Yaskawa INFORM job: SKRZYNIA_5140_180_STOPNI_10B_NEW.JBI

/JOB
//NAME SKRZYNIA_5140_180_STOPNI_10B_NEW
///FOLDERNAME 02-SKRZYNIE_JOBS
//POS
///NPOS 714,714,0,30,0,0
///TOOL 0
///POSTYPE PULSE
///PULSE
C00000=-21231,-51303,42314,2367,6591,-1439
C00001=-12854,-61498,-6635,149088,-29435,16513
C00002=84284,-61498,-6635,149088,14842,16513
C00003=84426,-61498,-62039,149088,14842,16513
C00004=84426,-61498,-83719,149088,14842,16513
C00005=40079,-25830,-61904,72398,37828,17494
C00006=40079,-25830,-61904,72398,37828,17494
C00007=38824,-23395,-60038,72349,38727,17731
C00008=41545,-22667,-59464,70826,37145,18191
C00009=40079,-25830,-61904,72398,37828,17494
C00010=40079,-23879,-31232,97616,36989,2612
C00011=40241,-22903,-30855,97033,36795,2952
C00012=39596,-21803,-29985,96678,37187,3182
C00013=41542,-21522,-29763,96797,35874,3054
C00014=40241,-22903,-30855,97033,36795,2952
C00015=44500,-22967,-34027,49689,40772,15208
C00016=44759,-21950,-33222,49364,40770,15399
C00017=43898,-20603,-32137,49608,41392,15289
C00018=45676,-20288,-31878,48567,40497,15854
C00019=44759,-21950,-33222,49364,40770,15399
C00020=50639,-31838,-53853,40430,42590,20636
C00021=47737,-42531,-47731,84740,46626,-3202
C00022=73324,-51450,-15857,136644,48513,-27329
C00023=28578,-31257,-33285,101874,54895,-3139
C00024=29101,-23166,-41439,93785,52323,3372
C00025=30342,-16402,-40775,90158,51109,6027
C00026=29555,-14242,-38855,90054,51607,6222
C00027=31304,-14182,-38798,89754,50458,6198
C00028=30342,-16402,-40775,90158,51109,6027
C00029=37840,-26567,-47806,97824,39338,5403
C00030=38314,-22656,-45541,96192,38787,6352
C00031=38740,-21749,-44817,95954,38481,6451
C00032=38106,-20505,-43805,95701,38856,6673
C00033=39920,-20274,-43616,95549,37666,6573
C00034=38740,-21749,-44817,95954,38481,6451
C00035=35154,-23288,-28184,89821,43405,2441
C00036=35403,-21021,-26397,89340,43215,2751
C00037=34678,-19569,-25213,89063,43699,2948
C00038=36545,-19419,-25091,89018,42427,2940
C00039=35403,-21021,-26397,89340,43215,2751
C00040=46673,-28267,-59493,36306,49500,22578
C00041=47298,-25083,-54483,36432,48421,22382
C00042=46134,-23276,-53085,36983,49197,22170
C00043=48093,-22778,-52692,35651,48513,22818
C00044=47298,-25083,-54483,36432,48421,22382
C00045=43000,-32780,-49011,53703,41088,15214
C00046=66148,-65994,-55487,105361,28212,-7739
C00047=66148,-65994,-55487,105361,28212,-7739
C00048=59848,-54778,-49507,133915,29212,-10807
C00049=45497,-38347,-41839,114412,32622,-465
C00050=46376,-32635,-46933,102993,29107,5780
C00051=46303,-28031,-46898,97061,28371,8976
C00052=45038,-26161,-45521,96183,29128,9541
C00053=46946,-25787,-45238,96120,27855,9431
C00054=46303,-28031,-46898,97061,28371,8976
C00055=45864,-17128,1685,129467,40696,-9274
C00056=46023,-15894,1830,128891,40053,-8896
C00057=45181,-14790,2774,128176,40341,-8535
C00058=46921,-14545,2986,129317,39465,-9073
C00059=45402,-17127,796,128656,40504,-8810
C00060=42828,-21985,-11573,106778,34538,-1929
C00061=43349,-21404,-11124,106831,34165,-1930
C00062=42250,-19876,-9917,105946,34757,-1485
C00063=44494,-19460,-9583,106781,33302,-1837
C00064=42797,-21858,-11474,106726,34550,-1903
C00065=42956,-14057,7354,88292,32197,-569
C00066=43438,-13569,7781,88275,31880,-510
C00067=42549,-12302,8904,87823,32462,-349
C00068=44721,-11883,9282,88161,31033,-316
C00069=42944,-14884,6642,88491,32210,-682
C00070=72417,-64226,-72669,53660,37323,27470
C00071=81480,-74508,-67932,111005,17511,3722
C00072=42492,-36415,-29790,92406,42740,11684
C00073=29699,-14901,-14062,86637,51249,15251
C00074=28921,-12904,-12269,86425,51786,15406
C00075=30978,-12767,-12144,86426,50380,15429
C00076=29506,-17416,-16239,86937,51377,15018
C00077=88410,-69609,-60867,139529,19008,-8209
C00078=82254,-59190,-37505,135829,26015,-2584
C00079=48709,-26647,-10027,118963,31871,904
C00080=44740,-24992,-19428,105622,30913,8023
C00081=35836,-10089,175,120717,54219,3716
C00082=33571,-11609,-5533,116057,52820,8482
C00083=32638,-9483,-3533,115639,53262,8773
C00084=34483,-9329,-3384,116184,52162,8425
C00085=33571,-11609,-5533,116057,52820,8482
C00086=29299,-14235,-8112,85858,51306,13749
C00087=30258,-13056,-7056,85778,50658,13854
C00088=29454,-11053,-5212,85557,51212,13988
C00089=31306,-10982,-5149,85624,49953,14016
C00090=30258,-13056,-7056,85778,50658,13854
C00091=44150,-27478,-14760,79983,38437,11062
C00092=60260,-41997,-20174,82745,25327,6782
C00093=62412,-62489,-12046,-12266,17816,34850
C00094=0,-52280,40443,0,6876,0
C00095=-681,-52632,38645,-5695,5489,-631
C00096=-17840,-61498,-6635,-149088,-29435,-16513
C00097=-84284,-61498,-6635,-149088,14842,-16513
C00098=-84426,-61498,-62039,-149088,14842,-16513
C00099=-84426,-61498,-83719,-149088,14842,-16513
C00100=-83351,-27062,-60322,-167360,37385,6517
C00101=-83351,-27062,-60322,-167360,37385,23281
C00102=-45097,-23850,-79932,-76262,26943,-22849
C00103=-48253,-15729,-73342,-71138,25693,-24842
C00104=-50302,-13076,-73239,-65836,25323,-27140
C00105=-49401,-11675,-71961,-66260,25816,-27133
C00106=-50608,-11574,-71867,-65226,25249,-27391
C00107=-49660,-13361,-73494,-66442,25615,-26975
C00108=-48242,-21102,-77802,-73044,25430,-23851
C00109=-42432,-29691,-46140,-101591,34194,-3953
C00110=-40467,-32259,-45349,-89481,35752,-6083
C00111=-35590,-22323,-38089,-87474,43148,-7978
C00112=-34853,-20780,-36847,-87247,43643,-8181
C00113=-37029,-20471,-36594,-86926,42180,-8224
C00114=-35503,-23333,-38886,-87700,43207,-7835
C00115=-41659,-25848,-37197,-61468,39541,-12344
C00116=-42019,-23363,-32043,-63110,38591,-11327
C00117=-41283,-22167,-31102,-63128,39154,-11341
C00118=-43189,-21868,-30866,-62281,38009,-11788
C00119=-40846,-25460,-35158,-62968,39555,-11455
C00120=-39561,-32409,-42051,-71473,38885,-9254
C00121=-88477,-67032,-53890,-125185,13082,17955
C00122=-90715,-66667,-50935,-152816,24533,28486
C00123=-30735,-26920,-32844,-95116,50209,-1071
C00124=-37180,-24683,-31930,-114741,47007,2943
C00125=-36407,-19634,-34656,-109847,45004,-453
C00126=-38352,-16604,-33863,-108521,43129,-1176
C00127=-37479,-14809,-32279,-108169,43576,-1482
C00128=-39395,-14487,-31992,-108361,42368,-1194
C00129=-37253,-18321,-35339,-108644,43916,-1187
C00130=-30948,-19486,-27368,-89515,49970,-2899
C00131=-32453,-17458,-25663,-89179,48933,-3088
C00132=-31896,-16151,-24534,-89028,49305,-3221
C00133=-33527,-16125,-24510,-88960,48196,-3202
C00134=-31291,-18911,-26892,-89421,49733,-2955
C00135=-32789,-14788,-10714,-75998,48642,-1904
C00136=-33953,-13481,-9550,-75758,47902,-2112
C00137=-33380,-12226,-8408,-75670,48319,-2157
C00138=-35020,-12164,-8351,-75529,47228,-2306
C00139=-33300,-14767,-10697,-75957,48300,-1949
C00140=-33300,-14767,-10697,-75957,48300,-1949
C00141=-33901,-13199,-7224,-76945,47663,-1266
C00142=-33178,-11617,-5779,-76815,48184,-1329
C00143=-35129,-11426,-5603,-76688,46886,-1497
C00144=-32900,-14718,-9841,-76444,48459,-1584
C00145=-46324,-38325,-53351,-48650,39022,-16558
C00146=-84678,-53272,-42524,-56273,5220,-14251
C00147=-79949,-57830,-54545,-43165,18800,-25262
C00148=-85199,-63426,-59279,-35356,8253,-25340
C00149=-43240,-40066,-69296,-76804,34492,-13950
C00150=-32352,-24302,-62495,-76398,48702,-17646
C00151=-33867,-19497,-59989,-74208,48202,-18898
C00152=-33043,-17469,-58279,-74274,48770,-19034
C00153=-35172,-17180,-58031,-73305,47532,-19251
C00154=-33150,-20833,-61090,-74721,48572,-18687
C00155=-32525,-19963,-22291,-97454,48417,-2656
C00156=-34479,-17146,-19937,-97221,47013,-2812
C00157=-33716,-15515,-18525,-96928,47480,-3025
C00158=-35357,-15455,-18472,-97073,46375,-2908
C00159=-33341,-18474,-21063,-97306,47817,-2759
C00160=-32838,-10388,7981,-94473,48357,2926
C00161=-33747,-9461,8037,-94117,47673,2571
C00162=-33094,-8062,9377,-93861,48090,2458
C00163=-34952,-7927,9507,-94260,46861,2543
C00164=-33010,-10379,7174,-94037,48174,2591
C00165=-36099,-20774,-22249,-70758,44565,-7624
C00166=-37926,-16067,-12890,-73276,42575,-5996
C00167=-37323,-14944,-11908,-73188,43017,-6038
C00168=-39053,-14785,-11769,-72915,41882,-6255
C00169=-37847,-19214,-17221,-72670,42783,-6386
C00170=-73757,-59015,-49060,-81128,17325,-3444
C00171=-66351,-49775,-22313,-134939,32824,19491
C00172=-38126,-18978,-6321,-103556,42156,4232
C00173=-39485,-17529,-8330,-90200,39091,223
C00174=-38315,-15563,-6658,-89669,39866,-39
C00175=-40130,-15376,-6497,-89855,38637,-21
C00176=-40610,-23081,-12745,-91737,38407,1092
C00177=-82794,-45547,-18103,-153793,26453,27163
C00178=-59391,-59726,-723,-139936,47315,26256
C00179=-59391,-63256,-7305,-138930,45803,25558
C00180=-41911,-25348,-18707,-96909,37821,5942
C00181=-39278,-18921,-13723,-94727,39374,4724
C00182=-50267,-3803,20766,-145166,53580,20077
C00183=-49199,-2294,22340,-144514,53890,19722
C00184=-50839,-1881,22778,-145489,53339,20243
C00185=-50267,-457,30009,-146420,56926,21139
C00186=-39278,-18921,-13723,-94727,39374,4724
C00187=-38355,-17353,-12416,-94258,39960,4466
C00188=-40180,-17161,-12255,-94505,38724,4557
C00189=-37963,-22229,-16363,-95272,40353,5112
C00190=-56568,-73357,-35482,-123268,35826,13545
C00191=-46099,-67236,-11725,-98004,28606,19827
C00192=275,-40498,62911,330,272,-175
C00193=-21231,-51303,42314,2367,6591,-1439
C00194=-12854,-61498,-6635,149088,-29435,16513
C00195=84284,-61498,-6635,149088,14842,16513
C00196=84426,-61498,-62039,149088,14842,16513
C00197=84426,-61498,-83719,149088,14842,16513
C00198=40079,-25830,-61904,72398,37828,17494
C00199=43542,-21744,-53414,85694,32141,12908
C00200=43538,-20959,-59091,78847,32551,16732
C00201=40079,-23879,-31232,97616,36989,2612
C00202=41069,-22296,-36683,87871,35939,7163
C00203=41069,-20857,-27994,94343,36275,3375
C00204=40241,-22903,-30855,97033,36795,2952
C00205=44500,-22967,-34027,49689,40772,15208
C00206=37674,-14410,-29425,54908,51799,12689
C00207=37617,-13106,-20810,58248,49229,10178
C00208=44759,-21950,-33222,49364,40770,15399
C00209=50639,-31838,-53853,40430,42590,20636
C00210=47737,-42531,-47731,84740,46626,-3202
C00211=78713,-49095,-28754,133607,38203,-24422
C00212=28578,-31257,-33285,101874,54895,-3139
C00213=29101,-23166,-41439,93785,52323,3372
C00214=31163,-13872,-34138,92103,50752,4440
C00215=31163,-14064,-41434,88282,50498,7326
C00216=30342,-16402,-40775,90158,51109,6027
C00217=37840,-26567,-47806,97824,39338,5403
C00218=38314,-22656,-45541,96192,38787,6352
C00219=39658,-19881,-39017,99036,38353,4498
C00220=39658,-20227,-46296,93241,37598,7980
C00221=38740,-21749,-44817,95954,38481,6451
C00222=35154,-23288,-28184,89821,43405,2441
C00223=36302,-20456,-32356,81251,42995,6506
C00224=36302,-19046,-24537,85721,42698,3608
C00225=35403,-21021,-26397,89340,43215,2751
C00226=46673,-28267,-59493,36306,49500,22578
C00227=35383,-14910,-45807,52457,59655,19882
C00228=35383,-15025,-38926,54776,56903,17744
C00229=47298,-25083,-54483,36432,48421,22382
C00230=43000,-32780,-49011,53703,41088,15214
C00231=90538,-65158,-52413,145953,6697,-22013
C00232=90538,-65158,-52413,145953,6697,-22013
C00233=59848,-54778,-49507,133915,29212,-10807
C00234=45497,-38347,-41839,114412,32622,-465
C00235=46376,-32635,-46933,102993,29107,5780
C00236=38443,-20223,-37840,96971,39567,10287
C00237=38443,-20698,-44956,91660,38993,13539
C00238=46303,-28031,-46898,97061,28371,8976
C00239=45864,-17128,1685,129467,40696,-9274
C00240=38069,-7942,12691,120284,49952,-5070
C00241=38069,-11604,1369,116685,47266,-2469
C00242=45402,-17127,796,128656,40504,-8810
C00243=42828,-21985,-11573,106778,34538,-1929
C00244=33281,-15275,-13406,92642,47209,4970
C00245=33281,-12456,-2996,97026,47894,1870
C00246=42797,-21858,-11474,106726,34550,-1903
C00247=42956,-14057,7354,88292,32197,-569
C00248=35915,-8349,8335,81338,43542,2014
C00249=35915,-4149,20758,86814,43229,-1568
C00250=42944,-14884,6642,88491,32210,-682
C00251=72417,-64226,-72669,53660,37323,27470
C00252=81480,-74508,-67932,111005,17511,3722
C00253=42492,-36415,-29790,92406,42740,11684
C00254=30589,-12517,-11440,90322,50747,14596
C00255=30928,-12247,-10742,85035,50377,15419
C00256=29506,-17416,-16239,86937,51377,15018
C00257=88410,-69609,-60867,139529,19008,-8209
C00258=82254,-59190,-37505,135829,26015,-2584
C00259=48709,-26647,-10027,118963,31871,904
C00260=44740,-24992,-19428,105622,30913,8023
C00261=35836,-10089,175,120717,54219,3716
C00262=34345,-8030,793,117331,53206,7509
C00263=34322,-10419,-8163,114502,51063,9720
C00264=33571,-11609,-5533,116057,52820,8482
C00265=29299,-14235,-8112,85858,51306,13749
C00266=31207,-11656,-8788,84025,50108,15207
C00267=31207,-8775,1760,88103,49995,12167
C00268=30258,-13056,-7056,85778,50658,13854
C00269=44150,-27478,-14760,79983,38437,11062
C00270=60260,-41997,-20174,82745,25327,6782
C00271=62412,-62489,-12046,-12266,17816,34850
C00272=0,-52280,40443,0,6876,0
C00273=-681,-52632,38645,-5695,5489,-631
C00274=-17840,-61498,-6635,-149088,-29435,-16513
C00275=-84284,-61498,-6635,-149088,14842,-16513
C00276=-84426,-61498,-62039,-149088,14842,-16513
C00277=-84426,-61498,-83719,-149088,14842,-16513
C00278=-83351,-27062,-60322,-167360,37385,6517
C00279=-83351,-27062,-60322,-167360,37385,23281
C00280=-45097,-23850,-79932,-76262,26943,-22849
C00281=-48253,-15729,-73342,-71138,25693,-24842
C00282=-42869,-6204,-67496,-75794,33821,-25861
C00283=-42869,-3205,-70686,-69723,34977,-29338
C00284=-49660,-13361,-73494,-66442,25615,-26975
C00285=-48242,-21102,-77802,-73044,25430,-23851
C00286=-42432,-29691,-46140,-101591,34194,-3953
C00287=-40467,-32259,-45349,-89481,35752,-6083
C00288=-32032,-15700,-34761,-86363,49905,-9645
C00289=-32032,-14866,-27372,-89947,49973,-6979
C00290=-35503,-23333,-38886,-87700,43207,-7835
C00291=-41659,-25848,-37197,-61468,39541,-12344
C00292=-32550,-13183,-23016,-68651,53358,-8526
C00293=-34023,-12481,-22084,-63241,53452,-9524
C00294=-40846,-25460,-35158,-62968,39555,-11455
C00295=-39561,-32409,-42051,-71473,38885,-9254
C00296=-88477,-67032,-53890,-125185,13082,17955
C00297=-90715,-66667,-50935,-152816,24533,28486
C00298=-30735,-26920,-32844,-95116,50209,-1071
C00299=-37180,-24683,-31930,-114741,47007,2943
C00300=-36407,-19634,-34656,-109847,45004,-453
C00301=-39264,-14095,-28560,-110319,43249,69
C00302=-39254,-14742,-35710,-105973,41627,-2729
C00303=-37253,-18321,-35339,-108644,43916,-1187
C00304=-30948,-19486,-27368,-89515,49970,-2899
C00305=-33188,-17217,-33290,-80523,49125,-7157
C00306=-33231,-16133,-25752,-84153,48705,-4513
C00307=-31291,-18911,-26892,-89421,49733,-2955
C00308=-32789,-14788,-10714,-75998,48642,-1904
C00309=-32456,-10000,-8763,-74569,51725,-2878
C00310=-32456,-7502,814,-78111,50801,-165
C00311=-33300,-14767,-10697,-75957,48300,-1949
C00312=-33300,-14767,-10697,-75957,48300,-1949
C00313=-31039,-7597,-4415,-75714,54029,-1891
C00314=-31745,-5891,1281,-74609,53027,-1007
C00315=-32900,-14718,-9841,-76444,48459,-1584
C00316=-46324,-38325,-53351,-48650,39022,-16558
C00317=-84678,-53272,-42524,-56273,5220,-14251
C00318=-79949,-57830,-54545,-43165,18800,-25262
C00319=-85199,-63426,-59279,-35356,8253,-25340
C00320=-43240,-40066,-69296,-76804,34492,-13950
C00321=-32352,-24302,-62495,-76398,48702,-17646
C00322=-34311,-15084,-43386,-89458,46770,-12174
C00323=-34303,-14562,-49859,-85086,46777,-15220
C00324=-33150,-20833,-61090,-74721,48572,-18687
C00325=-32525,-19963,-22291,-97454,48417,-2656
C00326=-35706,-13608,-12356,-102024,46946,-662
C00327=-35706,-15621,-21438,-97808,45877,-3577
C00328=-33341,-18474,-21063,-97306,47817,-2759
C00329=-32838,-10388,7981,-94473,48357,2926
C00330=-33093,-7396,5806,-90907,49596,566
C00331=-33114,-3922,16616,-94789,50065,3444
C00332=-33010,-10379,7174,-94037,48174,2591
C00333=-36099,-20774,-22249,-70758,44565,-7624
C00334=-34715,-11750,-12273,-72011,49148,-6727
C00335=-34715,-9605,-3694,-75523,48112,-4187
C00336=-37847,-19214,-17221,-72670,42783,-6386
C00337=-73757,-59015,-49060,-81128,17325,-3444
C00338=-66351,-49775,-22313,-134939,32824,19491
C00339=-38126,-18978,-6321,-103556,42156,4232
C00340=-35411,-10902,-672,-92816,45935,848
C00341=-36000,-11295,-2683,-84848,44809,-1301
C00342=-40610,-23081,-12745,-91737,38407,1092
C00343=-82794,-45547,-18103,-153793,26453,27163
C00344=-59391,-59726,-723,-139936,47315,26256
C00345=-59391,-69594,-18878,-137021,43274,24283
C00346=-41911,-25348,-18707,-96909,37821,5942
C00347=-39278,-18921,-13723,-94727,39374,4724
C00348=-41964,3488,28151,-134521,60914,14195
C00349=-41964,-819,15200,-132329,56719,12142
C00350=-50267,-457,30009,-146420,56926,21139
C00351=-33715,-10212,-1364,-94538,48612,5206
C00352=-33715,-12585,-10220,-90890,48191,2581
C00353=-37963,-22229,-16363,-95272,40353,5112
C00354=-66368,-73811,-34662,-141094,38161,28545
C00355=-46099,-67236,-11725,-98004,28606,19827
C00356=275,-40498,62911,330,272,-175
C00357=-21231,-51303,42314,2367,6591,-1439
C00358=-12854,-61498,-6635,149088,-29435,16513
C00359=32880,-72586,-50560,79734,53940,25582
C00360=76664,-93599,-96338,114349,24908,7990
C00361=72545,-76403,-90681,98079,12187,16258
C00362=68435,-42241,-79282,43384,21203,43145
C00363=65057,-16377,-54230,51764,24572,24912
C00364=65057,-16377,-54230,51764,24572,24912
C00365=63338,-14509,-52578,53100,25585,24479
C00366=65493,-13068,-51269,50530,24633,25485
C00367=65057,-16377,-54230,51764,24572,24912
C00368=65057,-15356,-24189,99795,20011,765
C00369=64877,-14372,-23690,98704,20045,1316
C00370=64002,-13489,-22890,98156,20604,1621
C00371=65592,-12702,-22173,98357,19527,1466
C00372=64877,-14372,-23690,98704,20045,1316
C00373=68341,-13254,-25781,29903,31229,25524
C00374=68283,-12212,-24821,29865,31356,25548
C00375=67188,-11145,-23825,30867,31841,25051
C00376=68624,-10377,-23095,29361,31405,25809
C00377=68283,-12212,-24821,29865,31356,25548
C00378=67373,-28813,-51747,26561,36937,27500
C00379=65665,-56911,-59086,75825,31170,1181
C00380=86238,-56758,-47218,93606,16664,-7096
C00381=86238,-56758,-47218,93606,16664,-7096
C00382=58162,-25487,-29222,106212,35121,-6052
C00383=54729,-17550,-36821,90686,35172,3055
C00384=53879,-10723,-35593,84994,35691,6442
C00385=52628,-8898,-33837,85063,36512,6546
C00386=54193,-8333,-33282,84633,35489,6620
C00387=53879,-10723,-35593,84994,35691,6442
C00388=63265,-18185,-41125,95483,22448,4389
C00389=62561,-14368,-38517,92984,22773,5727
C00390=62689,-13396,-37636,92694,22678,5861
C00391=61812,-12400,-36718,92465,23238,6064
C00392=63331,-11679,-36046,92201,22238,6052
C00393=62689,-13396,-37636,92694,22678,5861
C00394=60836,-16142,-22303,87853,25853,3109
C00395=60346,-13901,-20318,87240,26185,3441
C00396=59279,-12702,-19226,86999,26911,3593
C00397=60868,-12050,-18626,86765,25831,3679
C00398=60346,-13901,-20318,87240,26185,3441
C00399=71174,-16943,-50501,16787,44328,31924
C00400=70846,-13961,-45205,17496,43056,31510
C00401=69412,-12602,-43961,18675,43507,30969
C00402=70949,-11616,-43043,17320,43301,31610
C00403=70846,-13961,-45205,17496,43056,31510
C00404=66765,-25643,-43957,33958,30926,25005
C00405=89904,-51519,-74342,14421,36812,44678
C00406=59533,-60921,-66479,83565,41795,11392
C00407=74572,-27669,-34920,136415,14797,-11887
C00408=72479,-21736,-38943,108586,11547,1590
C00409=70901,-17325,-38411,94105,11830,8638
C00410=69318,-15905,-37172,92885,12849,9347
C00411=70820,-15051,-36412,92531,11846,9399
C00412=70901,-17325,-38411,94105,11830,8638
C00413=70927,-7523,10343,151197,29871,-19432
C00414=70517,-6236,10737,150221,29352,-18933
C00415=69462,-5331,11645,148944,29606,-18324
C00416=70849,-4645,12343,150548,29173,-19084
C00417=70402,-7634,9356,150158,29478,-18907
C00418=68660,-13051,-4106,122816,18275,-8999
C00419=68895,-12351,-3471,122899,18094,-9031
C00420=67458,-11121,-2337,120787,18802,-8043
C00421=69212,-10147,-1425,122703,17774,-8922
C00422=68590,-12934,-4000,122687,18305,-8939
C00423=67960,-5141,15741,92957,15720,-628
C00424=68207,-4523,16370,92944,15555,-601
C00425=67051,-3465,17460,92338,16311,-404
C00426=68762,-2475,18496,92897,15183,-531
C00427=68227,-5981,14898,93242,15553,-745
C00428=75423,-38775,-29488,68062,11357,11878
C00429=83800,-53438,-37305,103753,14733,-1265
C00430=84801,-45035,-34192,112697,15383,1107
C00431=73693,-37430,-30368,101200,21937,8332
C00432=54083,-9583,-9164,86048,34613,15862
C00433=52816,-7862,-7494,85864,35484,15962
C00434=54627,-7152,-6792,85763,34247,16030
C00435=54668,-12069,-11504,86415,34208,15656
C00436=89016,-59505,-36896,143842,20811,-11822
C00437=60495,-76741,-47652,120298,37447,-3273
C00438=76037,-16315,-2108,148598,17507,-12246
C00439=70560,-15452,-11753,122116,14270,428
C00440=59169,-3122,7113,131317,41741,-2292
C00441=57131,-5277,619,125436,39242,3005
C00442=55729,-3443,2508,124592,39934,3479
C00443=57337,-2775,3210,125461,39069,2998
C00444=57131,-5277,619,125436,39242,3005
C00445=54062,-9026,-3291,86300,34474,14396
C00446=54568,-7612,-1915,86151,34132,14497
C00447=53276,-5879,-187,85948,35014,14576
C00448=54919,-5291,406,85945,33897,14626
C00449=54568,-7612,-1915,86151,34132,14497
C00450=55516,-30048,-16468,81245,30784,11190
C00451=78642,-41617,-20006,83725,13431,8209
C00452=0,-52280,40443,0,6876,0
C00453=-681,-52632,38645,-5695,5489,-631
C00454=-17840,-61498,-6635,-149088,-29435,-16513
C00455=-84284,-61498,-6635,-149088,14842,-16513
C00456=-57949,-92832,-68327,-119114,39180,-13331
C00457=-51160,-78996,-68705,-103851,38676,-21739
C00458=-70129,-12201,-70194,-45988,15849,-32683
C00459=-70861,-4247,-62448,-43170,16032,-33903
C00460=-72229,-1292,-61598,-37253,16795,-36501
C00461=-71164,-286,-60510,-39045,17142,-35862
C00462=-72168,114,-60071,-37345,16819,-36474
C00463=-71747,-1710,-62044,-38091,16943,-36199
C00464=-72086,-8949,-67137,-41785,15362,-34318
C00465=-68226,-19972,-38714,-103620,16923,-1218
C00466=-67549,-22986,-38612,-80975,17520,-9124
C00467=-60286,-14955,-31870,-81576,26630,-9634
C00468=-59206,-13694,-30736,-81541,27366,-9725
C00469=-61026,-12796,-29913,-80837,26167,-9971
C00470=-60502,-15936,-32740,-81790,26471,-9505
C00471=-66711,-16726,-29834,-42060,26790,-21996
C00472=-66477,-14329,-24475,-44917,25565,-20507
C00473=-65503,-13376,-23611,-45716,26132,-20127
C00474=-67048,-12587,-22889,-44009,25442,-20959
C00475=-66009,-16611,-27996,-44380,26285,-20808
C00476=-67084,-23473,-35621,-52822,22843,-18344
C00477=-54372,-63877,-56403,-90862,27079,1323
C00478=-55608,-75012,-34654,-126966,55573,20814
C00479=-55608,-75012,-34654,-126966,55573,20814
C00480=-58069,-20780,-28125,-95622,31565,-134
C00481=-62818,-16895,-25617,-123146,31403,8811
C00482=-60301,-12189,-28106,-114654,29999,4030
C00483=-61167,-8731,-26593,-112607,28768,2985
C00484=-59960,-7252,-25135,-111997,29446,2563
C00485=-61574,-6413,-24296,-112502,28453,2957
C00486=-60636,-10677,-28466,-112685,29164,2987
C00487=-55814,-13636,-22293,-87541,33030,-3263
C00488=-56566,-11270,-20110,-87077,32519,-3496
C00489=-55709,-10167,-19066,-86969,33101,-3589
C00490=-57154,-9687,-18605,-86794,32120,-3632
C00491=-55949,-12989,-21706,-87412,32939,-3330
C00492=-57109,-8613,-4995,-71756,32687,-5152
C00493=-57764,-7017,-3429,-71410,32292,-5358
C00494=-56909,-5946,-2356,-71529,32873,-5273
C00495=-58347,-5433,-1836,-71115,31941,-5534
C00496=-57555,-8453,-4841,-71622,32398,-5235
C00497=-57555,-8453,-4841,-71622,32398,-5235
C00498=-57844,-6749,-1100,-73475,31868,-4209
C00499=-56760,-5394,262,-73573,32605,-4123
C00500=-58439,-4668,1002,-73167,31507,-4396
C00501=-57269,-8513,-4090,-72514,32435,-4729
C00502=-74194,-26905,-45748,-21164,30431,-30370
C00503=-93036,-61583,-83098,-4972,39040,-38907
C00504=-93036,-61583,-83098,-4972,39040,-38907
C00505=-71878,-28414,-61729,-48672,19032,-25171
C00506=-58025,-17185,-56692,-61796,34178,-22014
C00507=-58138,-12270,-53641,-59720,34855,-23185
C00508=-56898,-10637,-52111,-60384,35596,-23031
C00509=-58712,-9745,-51261,-58987,34681,-23500
C00510=-57851,-13714,-54968,-60141,34926,-22995
C00511=-57767,-13689,-16896,-100181,31334,-836
C00512=-58645,-10437,-13885,-99794,30663,-1040
C00513=-57513,-9065,-12573,-99347,31388,-1300
C00514=-58947,-8556,-12078,-99591,30423,-1148
C00515=-58031,-12031,-15383,-99926,31110,-974
C00516=-57646,-4162,14084,-101426,32077,4804
C00517=-58050,-2999,14481,-100683,31666,4357
C00518=-57067,-1784,15765,-100255,32298,4198
C00519=-58672,-1130,16464,-100866,31256,4407
C00520=-57676,-4116,13320,-100600,31921,4338
C00521=-61201,-13510,-16039,-60848,29053,-13371
C00522=-61885,-8475,-5914,-65722,27292,-10768
C00523=-61040,-7537,-4993,-65975,27855,-10622
C00524=-62506,-6917,-4380,-65230,26947,-11038
C00525=-62587,-11561,-10517,-63923,27184,-11731
C00526=-69972,-70945,-58827,-87515,19733,-17
C00527=-69972,-70945,-58827,-87515,19733,-17
C00528=-64053,-11295,342,-114563,25508,8776
C00529=-64305,-9514,-1154,-92513,22236,350
C00530=-62690,-7882,422,-91839,23314,70
C00531=-64201,-7220,1072,-92034,22288,112
C00532=-67149,-14673,-5883,-94845,20391,1413
C00533=-66017,-67071,-29713,-134523,32873,22112
C00534=-66017,-67071,-29713,-134523,48860,22112
C00535=-66017,-67071,-29713,-134523,48860,22112
C00536=-68464,-16512,-11702,-102583,19802,8050
C00537=-64069,-10918,-6685,-98748,22529,6223
C00538=-71808,7543,33524,-159735,48317,27747
C00539=-70546,8877,35161,-158835,48660,27285
C00540=-71854,9797,36309,-159820,48523,27800
C00541=-71808,11433,44144,-160620,52560,28413
C00542=-64069,-10918,-6685,-98748,22529,6223
C00543=-62794,-9626,-5461,-98007,23355,5872
C00544=-64311,-8958,-4821,-98397,22329,6039
C00545=-64031,-14482,-9933,-99750,22651,6736
C00546=-78219,-66180,-35295,-149347,29259,30999
C00547=-46099,-67236,-11725,-98004,28606,19827
C00548=275,-40498,62911,330,272,-175
C00549=-21231,-51303,42314,2367,6591,-1439
C00550=-12854,-61498,-6635,149088,-29435,16513
C00551=84284,-61498,-6635,149088,14842,16513
C00552=84426,-61498,-62039,149088,14842,16513
C00553=84426,-61498,-83719,149088,14842,16513
C00554=65057,-16377,-54230,51764,24572,24912
C00555=84197,-12836,-45810,-45141,8815,68584
C00556=84197,-12041,-51210,-30828,12194,61758
C00557=65057,-15356,-24189,99795,20011,765
C00558=74080,-15423,-30907,69143,7686,14038
C00559=74080,-14352,-23480,100923,7503,-991
C00560=64877,-14372,-23690,98704,20045,1316
C00561=68341,-13254,-25781,29903,31229,25524
C00562=74439,-11496,-26749,13621,29642,33649
C00563=74439,-10401,-19085,15788,25340,32499
C00564=68283,-12212,-24821,29865,31356,25548
C00565=75452,-19560,-44582,17787,36745,31835
C00566=68183,-44834,-62310,40554,34116,19994
C00567=94103,-63119,-69903,16230,17694,31762
C00568=91219,-55958,-51219,93435,14423,-1742
C00569=58162,-25487,-29222,106212,35121,-6052
C00570=54729,-17550,-36821,90686,35172,3055
C00571=70769,-15160,-35297,83470,11760,4000
C00572=70769,-15377,-40609,67973,12489,11436
C00573=53879,-10723,-35593,84994,35691,6442
C00574=63265,-18185,-41125,95483,22448,4389
C00575=62561,-14368,-38517,92984,22773,5727
C00576=77715,-13962,-33882,144680,4496,-21400
C00577=77806,-14046,-41277,60589,2532,18064
C00578=62689,-13396,-37636,92694,22678,5861
C00579=60836,-16142,-22303,87853,25853,3109
C00580=74678,-16514,-29029,42946,9451,23276
C00581=74678,-15315,-21920,65026,7151,12815
C00582=60346,-13901,-20318,87240,26185,3441
C00583=71174,-16943,-50501,16787,44328,31924
C00584=80494,-13102,-44599,-1731,38384,44653
C00585=80494,-13295,-38861,-1907,34285,44756
C00586=70846,-13961,-45205,17496,43056,31510
C00587=69645,-22678,-41665,30358,30421,26767
C00588=81017,-78801,-66317,80675,7786,2447
C00589=81017,-78801,-66317,80675,7786,2447
C00590=74572,-27669,-34920,136415,14797,-11887
C00591=72479,-21736,-38943,108586,11547,1590
C00592=76162,-15538,-34076,119407,5153,-4143
C00593=76225,-15803,-40874,66675,4586,20654
C00594=70901,-17325,-38411,94105,11830,8638
C00595=70927,-7523,10343,151197,29871,-19432
C00596=75273,-951,23395,164730,33684,-27271
C00597=75257,-4812,11918,163197,28775,-26429
C00598=70402,-7634,9356,150158,29478,-18907
C00599=68660,-13051,-4106,122816,18275,-8999
C00600=75422,-13779,-12311,124767,7049,-10125
C00601=75402,-11409,-3274,143452,10422,-18986
C00602=68590,-12934,-4000,122687,18305,-8939
C00603=67960,-5141,15741,92957,15720,-628
C00604=77005,-5383,11265,73049,3770,10304
C00605=77005,-1367,23224,135174,5603,-18901
C00606=68227,-5981,14898,93242,15553,-745
C00607=83595,-66668,-34414,154325,14846,-28455
C00608=83595,-66668,-34414,154325,14846,-28455
C00609=69137,-30288,-25983,94330,24536,11676
C00610=73329,-13700,-12516,109108,8203,5807
C00611=73329,-11353,-3574,130600,10679,-4409
C00612=54668,-12069,-11504,86415,34208,15656
C00613=46050,-47732,-32699,100114,41423,7030
C00614=72866,-68602,-36981,132032,32409,-7906
C00615=72866,-68602,-36981,132032,32409,-7906
C00616=76037,-16315,-2108,148598,17507,-12246
C00617=70560,-15452,-11753,122116,14270,428
C00618=59169,-3122,7113,131317,41741,-2292
C00619=72693,-1568,14493,161814,36543,-14367
C00620=75650,3978,23428,169507,44505,-15919
C00621=70596,-8585,4037,153028,29768,-12051
C00622=54062,-9026,-3291,86300,34474,14396
C00623=70728,-11880,-8994,79432,11308,18593
C00624=70728,-9344,357,101276,11563,8141
C00625=54568,-7612,-1915,86151,34132,14497
C00626=62643,-28068,-15160,80125,26114,12294
C00627=92151,-29067,-13111,41177,6909,29587
C00628=79691,-50270,-13176,-792,17881,39424
C00629=0,-52280,40443,0,6876,0
C00630=-681,-52632,38645,-5695,5489,-631
C00631=-17840,-61498,-6635,-149088,-29435,-16513
C00632=-84284,-61498,-6635,-149088,14842,-16513
C00633=-84426,-61498,-62039,-149088,14842,-16513
C00634=-84426,-61498,-83719,-149088,14842,-16513
C00635=-83351,-27062,-60322,-167360,37385,6517
C00636=-83351,-27062,-60322,-167360,37385,23281
C00637=-70129,-12201,-70194,-45988,15849,-32683
C00638=-70861,-4247,-62448,-43170,16032,-33903
C00639=-76882,43,-60950,-14294,14755,-45201
C00640=-76882,3984,-64926,-10429,20329,-47102
C00641=-71747,-1710,-62044,-38091,16943,-36199
C00642=-72086,-8949,-67137,-41785,15362,-34318
C00643=-68226,-19972,-38714,-103620,16923,-1218
C00644=-67549,-22986,-38612,-80975,17520,-9124
C00645=-69143,-15166,-34287,-68804,15212,-14794
C00646=-69143,-14592,-28782,-80821,14459,-8960
C00647=-60502,-15936,-32740,-81790,26471,-9505
C00648=-66711,-16726,-29834,-42060,26790,-21996
C00649=-75652,-13136,-22972,-17539,18443,-33643
C00650=-76393,-11602,-18975,-13556,19574,-34543
C00651=-66009,-16611,-27996,-44380,26285,-20808
C00652=-61601,-28306,-39228,-59626,25389,-15050
C00653=-72315,-63222,-70224,-69600,33305,-10426
C00654=-72315,-63222,-70224,-69600,33305,-10426
C00655=-58069,-20780,-28125,-95622,31565,-134
C00656=-62818,-16895,-25617,-123146,31403,8811
C00657=-60301,-12189,-28106,-114654,29999,4030
C00658=-75089,-9933,-24682,-148597,14783,22922
C00659=-75089,-10642,-34451,-132584,9653,15243
C00660=-60636,-10677,-28466,-112685,29164,2987
C00661=-55814,-13636,-22293,-87541,33030,-3263
C00662=-73301,-16058,-32281,-44459,12702,-22095
C00663=-73339,-15052,-25249,-60236,10249,-14543
C00664=-55949,-12989,-21706,-87412,32939,-3330
C00665=-57109,-8613,-4995,-71756,32687,-5152
C00666=-71674,-10355,-9102,-48278,15013,-17468
C00667=-71670,-8088,-356,-62615,12652,-10541
C00668=-57555,-8453,-4841,-71622,32398,-5235
C00669=-57555,-8453,-4841,-71622,32398,-5235
C00670=-73349,-10209,-7254,-46090,12597,-18565
C00671=-73349,-7867,1452,-63091,10217,-10432
C00672=-57269,-8513,-4090,-72514,32435,-4729
C00673=-74194,-26905,-45748,-21164,30431,-30370
C00674=-76007,-77202,-67157,-59280,11041,-11579
C00675=-76006,-77203,-67157,-59281,11043,-11581
C00676=-53398,-42726,-55849,-45492,34374,-18069
C00677=-71878,-28414,-61729,-48672,19032,-25171
C00678=-58025,-17185,-56692,-61796,34178,-22014
C00679=-77553,-14661,-43008,-35465,5780,-31120
C00680=-77553,-14004,-50514,-17997,10868,-39389
C00681=-57851,-13714,-54968,-60141,34926,-22995
C00682=-57767,-13689,-16896,-100181,31334,-836
C00683=-74769,-11126,-10073,-142523,13426,19686
C00684=-74753,-12848,-17783,-130765,10301,14051
C00685=-58031,-12031,-15383,-99926,31110,-974
C00686=-57646,-4162,14084,-101426,32077,4804
C00687=-72179,-7124,6017,-115427,12582,9833
C00688=-72179,-4103,15503,-129018,15105,16401
C00689=-57676,-4116,13320,-100600,31921,4338
C00690=-61201,-13510,-16039,-60848,29053,-13371
C00691=-74136,-10643,-11909,-32993,14820,-27251
C00692=-74162,-8377,-2780,-45377,11297,-21290
C00693=-62587,-11561,-10517,-63923,27184,-11731
C00694=-68334,-63389,-52515,-83837,20864,-1739
C00695=-68334,-63389,-52515,-83837,20864,-1739
C00696=-64053,-11295,342,-114563,25508,8776
C00697=-75758,-9453,-2048,-123101,7379,13416
C00698=-76003,-8378,955,-106758,5948,6887
C00699=-67149,-14673,-5883,-94845,20391,1413
C00700=-65551,-48104,-28924,-114827,24376,11665
C00701=-39771,-60653,-24362,-111239,58263,14171
C00702=-39771,-60652,-24363,-111239,58260,14167
C00703=-68464,-16512,-11702,-102583,19802,8050
C00704=-64069,-10918,-6685,-98748,22529,6223
C00705=-75794,5019,20382,-166088,42002,32193
C00706=-75794,5019,20382,-166088,42002,32193
C00707=-71808,11433,44144,-160620,52560,28413
C00708=-74529,-9237,-439,-131085,10959,21329
C00709=-74560,-11298,-8213,-120962,9324,16064
C00710=-64031,-14482,-9933,-99750,22651,6736
C00711=-65667,-47452,-26760,-125785,27682,20101
C00712=-46099,-67236,-11725,-98004,28606,19827
C00713=275,-40498,62911,330,272,-175
BC00000=467225
BC00001=513669
BC00002=494109
BC00003=467540
BC00004=467540
BC00005=478876
BC00006=478876
BC00007=478876
BC00008=478876
BC00009=478876
BC00010=478876
BC00011=478876
BC00012=478876
BC00013=478876
BC00014=478876
BC00015=478876
BC00016=478876
BC00017=478876
BC00018=478876
BC00019=478876
BC00020=478876
BC00021=481980
BC00022=563952
BC00023=606256
BC00024=606256
BC00025=606252
BC00026=606252
BC00027=606252
BC00028=606252
BC00029=654662
BC00030=654618
BC00031=654618
BC00032=654618
BC00033=654618
BC00034=654618
BC00035=654618
BC00036=654618
BC00037=654618
BC00038=654618
BC00039=654618
BC00040=686402
BC00041=686402
BC00042=686350
BC00043=686350
BC00044=686402
BC00045=652574
BC00046=648164
BC00047=761837
BC00048=784046
BC00049=784046
BC00050=784046
BC00051=784046
BC00052=784046
BC00053=784046
BC00054=784046
BC00055=784046
BC00056=784046
BC00057=784046
BC00058=784046
BC00059=784046
BC00060=821134
BC00061=821134
BC00062=821134
BC00063=821134
BC00064=821134
BC00065=821134
BC00066=821134
BC00067=821134
BC00068=821134
BC00069=821134
BC00070=849627
BC00071=945583
BC00072=909600
BC00073=909600
BC00074=909600
BC00075=909600
BC00076=909600
BC00077=945583
BC00078=1005127
BC00079=999652
BC00080=999652
BC00081=991093
BC00082=990930
BC00083=990930
BC00084=990930
BC00085=990930
BC00086=990930
BC00087=990930
BC00088=990930
BC00089=990930
BC00090=990930
BC00091=981572
BC00092=972138
BC00093=892453
BC00094=828403
BC00095=518986
BC00096=509920
BC00097=467540
BC00098=467540
BC00099=467540
BC00100=521167
BC00101=520352
BC00102=535759
BC00103=535759
BC00104=535757
BC00105=535757
BC00106=535757
BC00107=535757
BC00108=535757
BC00109=485653
BC00110=485653
BC00111=485653
BC00112=485653
BC00113=485653
BC00114=485653
BC00115=485653
BC00116=485653
BC00117=485653
BC00118=485653
BC00119=485653
BC00120=485653
BC00121=485653
BC00122=615112
BC00123=615112
BC00124=615112
BC00125=615112
BC00126=615112
BC00127=615112
BC00128=615112
BC00129=615112
BC00130=615112
BC00131=615112
BC00132=615112
BC00133=615112
BC00134=615112
BC00135=615112
BC00136=615112
BC00137=615112
BC00138=615112
BC00139=615112
BC00140=658076
BC00141=658076
BC00142=658076
BC00143=658076
BC00144=658076
BC00145=655680
BC00146=643721
BC00147=643721
BC00148=793396
BC00149=799070
BC00150=799070
BC00151=799070
BC00152=799070
BC00153=799070
BC00154=799070
BC00155=799070
BC00156=799070
BC00157=799070
BC00158=799070
BC00159=799070
BC00160=799070
BC00161=799070
BC00162=799070
BC00163=799070
BC00164=799070
BC00165=845667
BC00166=845667
BC00167=845667
BC00168=845667
BC00169=845667
BC00170=845667
BC00171=899436
BC00172=899436
BC00173=899436
BC00174=899436
BC00175=899436
BC00176=899436
BC00177=899436
BC00178=862979
BC00179=977267
BC00180=1008066
BC00181=1008066
BC00182=995068
BC00183=995068
BC00184=995068
BC00185=995068
BC00186=1008066
BC00187=1008066
BC00188=1008066
BC00189=1008066
BC00190=991691
BC00191=895479
BC00192=639407
BC00193=467225
BC00194=513669
BC00195=494109
BC00196=467540
BC00197=467540
BC00198=478876
BC00199=478876
BC00200=478876
BC00201=478876
BC00202=478876
BC00203=478876
BC00204=478876
BC00205=478876
BC00206=478876
BC00207=478876
BC00208=478876
BC00209=478876
BC00210=481980
BC00211=563952
BC00212=606256
BC00213=606256
BC00214=606252
BC00215=606252
BC00216=606252
BC00217=654662
BC00218=654618
BC00219=654618
BC00220=654618
BC00221=654618
BC00222=654618
BC00223=654618
BC00224=654618
BC00225=654618
BC00226=686402
BC00227=686402
BC00228=686402
BC00229=686402
BC00230=652574
BC00231=641414
BC00232=715810
BC00233=784046
BC00234=784046
BC00235=784046
BC00236=784046
BC00237=784046
BC00238=784046
BC00239=784046
BC00240=784043
BC00241=784043
BC00242=784046
BC00243=821134
BC00244=821134
BC00245=821134
BC00246=821134
BC00247=821134
BC00248=821134
BC00249=821134
BC00250=821134
BC00251=849627
BC00252=945583
BC00253=909600
BC00254=909600
BC00255=909600
BC00256=909600
BC00257=945583
BC00258=1005127
BC00259=999652
BC00260=999652
BC00261=991093
BC00262=990930
BC00263=990930
BC00264=990930
BC00265=990930
BC00266=990930
BC00267=990930
BC00268=990930
BC00269=981572
BC00270=972138
BC00271=892453
BC00272=828403
BC00273=518986
BC00274=509920
BC00275=467540
BC00276=467540
BC00277=467540
BC00278=521167
BC00279=520352
BC00280=535759
BC00281=535759
BC00282=535757
BC00283=535757
BC00284=535757
BC00285=535757
BC00286=485653
BC00287=485653
BC00288=485653
BC00289=485653
BC00290=485653
BC00291=485653
BC00292=485653
BC00293=485653
BC00294=485653
BC00295=485653
BC00296=485653
BC00297=615112
BC00298=615112
BC00299=615112
BC00300=615112
BC00301=615112
BC00302=615112
BC00303=615112
BC00304=615112
BC00305=615112
BC00306=615112
BC00307=615112
BC00308=615112
BC00309=615112
BC00310=615112
BC00311=615112
BC00312=658076
BC00313=658076
BC00314=658076
BC00315=658076
BC00316=655680
BC00317=643721
BC00318=643721
BC00319=793396
BC00320=799070
BC00321=799070
BC00322=799070
BC00323=799070
BC00324=799070
BC00325=799070
BC00326=799070
BC00327=799070
BC00328=799070
BC00329=799070
BC00330=799070
BC00331=799070
BC00332=799070
BC00333=845667
BC00334=845667
BC00335=845667
BC00336=845667
BC00337=845667
BC00338=899436
BC00339=899436
BC00340=899436
BC00341=899436
BC00342=899436
BC00343=899436
BC00344=862979
BC00345=977267
BC00346=1008066
BC00347=1008066
BC00348=995068
BC00349=995068
BC00350=995068
BC00351=1008066
BC00352=1008066
BC00353=1008066
BC00354=1008066
BC00355=895479
BC00356=639407
BC00357=467225
BC00358=513669
BC00359=542621
BC00360=535309
BC00361=478364
BC00362=478364
BC00363=478876
BC00364=478876
BC00365=478876
BC00366=478876
BC00367=478876
BC00368=478876
BC00369=478876
BC00370=478876
BC00371=478876
BC00372=478876
BC00373=478876
BC00374=478876
BC00375=478876
BC00376=478876
BC00377=478876
BC00378=478876
BC00379=480759
BC00380=480759
BC00381=560395
BC00382=606256
BC00383=606256
BC00384=606252
BC00385=606252
BC00386=606252
BC00387=606252
BC00388=654662
BC00389=654618
BC00390=654618
BC00391=654618
BC00392=654618
BC00393=654618
BC00394=654618
BC00395=654618
BC00396=654618
BC00397=654618
BC00398=654618
BC00399=686402
BC00400=686402
BC00401=686350
BC00402=686350
BC00403=686402
BC00404=652574
BC00405=652574
BC00406=774850
BC00407=784046
BC00408=784046
BC00409=784046
BC00410=784046
BC00411=784046
BC00412=784046
BC00413=784046
BC00414=784046
BC00415=784046
BC00416=784046
BC00417=784046
BC00418=821134
BC00419=821134
BC00420=821134
BC00421=821134
BC00422=821134
BC00423=821134
BC00424=821134
BC00425=821134
BC00426=821134
BC00427=821134
BC00428=821134
BC00429=846623
BC00430=894838
BC00431=909600
BC00432=909600
BC00433=909600
BC00434=909600
BC00435=909600
BC00436=909600
BC00437=995060
BC00438=999652
BC00439=999652
BC00440=991093
BC00441=990930
BC00442=990930
BC00443=990930
BC00444=990930
BC00445=990930
BC00446=990930
BC00447=990930
BC00448=990930
BC00449=990930
BC00450=981572
BC00451=972138
BC00452=828403
BC00453=518986
BC00454=509920
BC00455=467540
BC00456=497868
BC00457=497868
BC00458=535759
BC00459=535759
BC00460=535757
BC00461=535757
BC00462=535757
BC00463=535757
BC00464=535757
BC00465=485653
BC00466=485653
BC00467=485653
BC00468=485653
BC00469=485653
BC00470=485653
BC00471=485653
BC00472=485653
BC00473=485653
BC00474=485653
BC00475=485653
BC00476=485653
BC00477=485653
BC00478=485653
BC00479=601945
BC00480=615112
BC00481=615112
BC00482=615112
BC00483=615112
BC00484=615112
BC00485=615112
BC00486=615112
BC00487=615112
BC00488=615112
BC00489=615112
BC00490=615112
BC00491=615112
BC00492=615112
BC00493=615112
BC00494=615112
BC00495=615112
BC00496=615112
BC00497=658076
BC00498=658076
BC00499=658076
BC00500=658076
BC00501=658076
BC00502=655680
BC00503=655680
BC00504=765678
BC00505=799070
BC00506=799070
BC00507=799070
BC00508=799070
BC00509=799070
BC00510=799070
BC00511=799070
BC00512=799070
BC00513=799070
BC00514=799070
BC00515=799070
BC00516=799070
BC00517=799070
BC00518=799070
BC00519=799070
BC00520=799070
BC00521=845667
BC00522=845667
BC00523=845667
BC00524=845667
BC00525=845667
BC00526=845667
BC00527=900547
BC00528=899436
BC00529=899436
BC00530=899436
BC00531=899436
BC00532=899436
BC00533=899436
BC00534=943124
BC00535=971560
BC00536=1008066
BC00537=1008066
BC00538=995068
BC00539=995068
BC00540=995068
BC00541=995068
BC00542=1008066
BC00543=1008066
BC00544=1008066
BC00545=1008066
BC00546=1008066
BC00547=895479
BC00548=639407
BC00549=467225
BC00550=513669
BC00551=494109
BC00552=467540
BC00553=467540
BC00554=478876
BC00555=478876
BC00556=478876
BC00557=478876
BC00558=478876
BC00559=478876
BC00560=478876
BC00561=478876
BC00562=478876
BC00563=478876
BC00564=478876
BC00565=478876
BC00566=479530
BC00567=502776
BC00568=571156
BC00569=606256
BC00570=606256
BC00571=606252
BC00572=606252
BC00573=606252
BC00574=654662
BC00575=654618
BC00576=654618
BC00577=654618
BC00578=654618
BC00579=654618
BC00580=654618
BC00581=654618
BC00582=654618
BC00583=686402
BC00584=686402
BC00585=686402
BC00586=686402
BC00587=652574
BC00588=654591
BC00589=763025
BC00590=784046
BC00591=784046
BC00592=784046
BC00593=784046
BC00594=784046
BC00595=784046
BC00596=784043
BC00597=784043
BC00598=784046
BC00599=821134
BC00600=821134
BC00601=821134
BC00602=821134
BC00603=821134
BC00604=821134
BC00605=821134
BC00606=821134
BC00607=821134
BC00608=884766
BC00609=909600
BC00610=909600
BC00611=909600
BC00612=909600
BC00613=909600
BC00614=909600
BC00615=972020
BC00616=999652
BC00617=999652
BC00618=991093
BC00619=990930
BC00620=990930
BC00621=990930
BC00622=990930
BC00623=990930
BC00624=990930
BC00625=990930
BC00626=981572
BC00627=972138
BC00628=920868
BC00629=828403
BC00630=518986
BC00631=509920
BC00632=467540
BC00633=467540
BC00634=467540
BC00635=521167
BC00636=520352
BC00637=535759
BC00638=535759
BC00639=535757
BC00640=535757
BC00641=535757
BC00642=535757
BC00643=485653
BC00644=485653
BC00645=485653
BC00646=485653
BC00647=485653
BC00648=485653
BC00649=485653
BC00650=485653
BC00651=485653
BC00652=485653
BC00653=485653
BC00654=600333
BC00655=615112
BC00656=615112
BC00657=615112
BC00658=615112
BC00659=615112
BC00660=615112
BC00661=615112
BC00662=615112
BC00663=615112
BC00664=615112
BC00665=615112
BC00666=615112
BC00667=615112
BC00668=615112
BC00669=658076
BC00670=658076
BC00671=658076
BC00672=658076
BC00673=655680
BC00674=656245
BC00675=762546
BC00676=762546
BC00677=799070
BC00678=799070
BC00679=799070
BC00680=799070
BC00681=799070
BC00682=799070
BC00683=799070
BC00684=799070
BC00685=799070
BC00686=799070
BC00687=799070
BC00688=799070
BC00689=799070
BC00690=845667
BC00691=845667
BC00692=845667
BC00693=845667
BC00694=845667
BC00695=902133
BC00696=899436
BC00697=899436
BC00698=899436
BC00699=899436
BC00700=899436
BC00701=899436
BC00702=981307
BC00703=1008066
BC00704=1008066
BC00705=1008527
BC00706=1000335
BC00707=995068
BC00708=1008066
BC00709=1008066
BC00710=1008066
BC00711=1008066
BC00712=895479
BC00713=639407
///POSTYPE BASE
///RECTAN
///RCONF 0,0,0,0,0,0,0,0,0,0,0,0,0,0,0,0,0,0,0,0,0,0,0,0
P00006=-2.449,0.031,8.825,0.0000,0.0000,0.0000
P00056=0.000,0.000,5.000,0.0000,0.0000,0.0000
P00301=0.005,-4.708,-4.628,0.0000,0.0000,0.0000
P00302=0.052,-2.937,-4.426,0.0000,0.0000,0.0000
P00303=-0.004,-1.437,-4.584,0.0000,0.0000,0.0000
P00304=0.028,-1.666,-4.234,0.0000,0.0000,0.0000
P00305=-0.003,-1.920,-3.501,0.0000,0.0000,0.0000
P00306=0.015,-2.252,-3.054,0.0000,0.0000,0.0000
P00307=0.019,-2.151,-5.077,0.0000,0.0000,0.0000
P00308=-0.003,-2.092,-4.888,0.0000,0.0000,0.0000
P00309=-0.040,-2.205,-4.992,0.0000,0.0000,0.0000
P00310=-0.006,-2.490,-5.925,0.0000,0.0000,0.0000
P00311=-0.007,-2.079,-5.307,0.0000,0.0000,0.0000
P00312=-0.032,2.202,-7.632,0.0000,0.0000,0.0000
///RCONF 1,0,0,0,0,0,0,0,0,0,0,0,0,0,0,0,0,0,0,0,0,0,0,0
P00313=-0.088,1.055,2.110,0.0000,0.0000,0.0000
P00314=-0.055,1.752,1.634,0.0000,0.0000,0.0000
///RCONF 0,0,0,0,0,0,0,0,0,0,0,0,0,0,0,0,0,0,0,0,0,0,0,0
P00351=13.563,-0.027,-0.653,0.0000,0.0000,0.0000
P00352=13.252,-0.027,-0.827,0.0000,0.0000,0.0000
P00353=10.971,-0.082,0.776,0.0000,0.0000,0.0000
P00354=-0.024,2.508,-1.824,0.0000,0.0000,0.0000
P00355=-0.001,2.528,-1.131,0.0000,0.0000,0.0000
P00356=-0.034,2.921,-0.262,0.0000,0.0000,0.0000
P00357=0.003,3.386,-0.091,0.0000,0.0000,0.0000
P00358=0.014,3.037,-0.020,0.0000,0.0000,0.0000
P00359=-0.005,2.731,0.912,0.0000,0.0000,0.0000
P00360=-0.011,3.412,0.438,0.0000,0.0000,0.0000
P00361=0.018,3.050,1.253,0.0000,0.0000,0.0000
P00362=0.014,2.784,0.148,0.0000,0.0000,0.0000
P00363=0.026,4.310,-2.639,0.0000,0.0000,0.0000
P00364=0.034,4.181,-4.040,0.0000,0.0000,0.0000
//INST
///DATE 2024/09/19 14:26
///ATTR SC,RW
///GROUP1 RB1,BS1
NOP
CALL JOB:MOVE_INTO_TUNNEL
MOVJ C00000 BC00000 VJ=10.00
MOVJ C00001 BC00001 VJ=10.00
MOVJ C00002 BC00002 VJ=10.00
MOVJ C00003 BC00003 VJ=10.00
MOVJ C00004 BC00004 VJ=10.00
'------------------------
'W29.2
'------------------------
MOVL C00005 BC00005 V=500.0
'------------------------
'W63.5
'------------------------
SFTOF
MOVL C00006 BC00006 V=166.7 PL=0
REFP 3 C00007 BC00007
CALL JOB:SEARCH-R1
IMOV P0056 V=50.0 PL=0
SET P0301 P0006
SFTON P0301
REFP 3 C00008 BC00008
CALL JOB:SEARCH-R1
SET P0301 P0006
SFTON P0301
MOVL C00009 BC00009 V=166.7 PL=0
SFTOF
MOVL C00010 BC00010 V=500.0
MOVL C00011 BC00011 V=166.7 PL=0
REFP 3 C00012 BC00012
CALL JOB:SEARCH-R1
IMOV P0056 V=50.0 PL=0
SET P0302 P0006
SFTON P0302
REFP 3 C00013 BC00013
CALL JOB:SEARCH-R1
SET P0302 P0006
SFTON P0302
MOVL C00014 BC00014 V=166.7 PL=0
SFTOF
MOVL C00015 BC00015 V=500.0
MOVL C00016 BC00016 V=166.7 PL=0
REFP 3 C00017 BC00017
CALL JOB:SEARCH-R1
IMOV P0056 V=50.0 PL=0
SET P0303 P0006
SFTON P0303
REFP 3 C00018 BC00018
CALL JOB:SEARCH-R1
SET P0303 P0006
SFTON P0303
SFTOF
MOVL C00019 BC00019 V=166.7 PL=0
MOVL C00020 BC00020 V=500.0
MOVJ C00021 BC00021 VJ=30.00
MOVJ C00022 BC00022 VJ=30.00
MOVJ C00023 BC00023 VJ=30.00
MOVL C00024 BC00024 V=500.0
'------------------------
'W29.14
'------------------------
MOVL C00025 BC00025 V=166.7 PL=0
REFP 3 C00026 BC00026
CALL JOB:SEARCH-R1
IMOV P0056 V=23.0 PL=0
SET P0304 P0006
SFTON P0304
REFP 3 C00027 BC00027
CALL JOB:SEARCH-R1
SET P0304 P0006
SFTON P0304
MOVL C00028 BC00028 V=66.7 PL=0
SFTOF
'PRZEJAZD
MOVL C00029 BC00029 V=500.0
MOVL C00030 BC00030 V=500.0
'------------------------
'W63.17
'------------------------
MOVL C00031 BC00031 V=166.7 PL=0
REFP 3 C00032 BC00032
CALL JOB:SEARCH-R1
IMOV P0056 V=23.0 PL=0
SET P0305 P0006
SFTON P0305
REFP 3 C00033 BC00033
CALL JOB:SEARCH-R1
SET P0305 P0006
SFTON P0305
MOVL C00034 BC00034 V=166.7 PL=0
SFTOF
MOVL C00035 BC00035 V=500.0
MOVL C00036 BC00036 V=166.7
REFP 3 C00037 BC00037
CALL JOB:SEARCH-R1
IMOV P0056 V=23.0 PL=0
SET P0306 P0006
SFTON P0306
REFP 3 C00038 BC00038
CALL JOB:SEARCH-R1
SET P0306 P0006
SFTON P0306
MOVL C00039 BC00039 V=166.7 PL=0
'PRZEJAZD
MOVL C00040 BC00040 V=500.0
MOVL C00041 BC00041 V=166.7
REFP 3 C00042 BC00042
CALL JOB:SEARCH-R1
IMOV P0056 V=23.0 PL=0
SET P0307 P0006
SFTON P0307
REFP 3 C00043 BC00043
CALL JOB:SEARCH-R1
SET P0307 P0006
SFTON P0307
MOVL C00044 BC00044 V=166.7 PL=0
SFTOF
MOVJ C00045 BC00045 VJ=20.00
MOVJ C00046 BC00046 VJ=20.00
MOVJ C00047 BC00047 VJ=30.00
MOVJ C00048 BC00048 VJ=30.00
MOVJ C00049 BC00049 VJ=30.00
MOVL C00050 BC00050 V=500.0
'------------------------
'W63.20
'------------------------
MOVL C00051 BC00051 V=166.7 PL=0
REFP 3 C00052 BC00052
CALL JOB:SEARCH-R1
IMOV P0056 V=23.0 PL=0
SET P0308 P0006
SFTON P0308
REFP 3 C00053 BC00053
CALL JOB:SEARCH-R1
SET P0308 P0006
SFTON P0308
MOVL C00054 BC00054 V=166.7 PL=0
SFTOF
'PRZEJAZD
MOVL C00055 BC00055 V=500.0
'------------------------
'W63.23
'------------------------
MOVL C00056 BC00056 V=166.7 PL=0
REFP 3 C00057 BC00057
CALL JOB:SEARCH-R1
IMOV P0056 V=23.0 PL=0
SET P0309 P0006
SFTON P0309
REFP 3 C00058 BC00058
CALL JOB:SEARCH-R1
SET P0309 P0006
SFTON P0309
MOVL C00059 BC00059 V=250.0 PL=0
SFTOF
MOVL C00060 BC00060 V=500.0
MOVL C00061 BC00061 V=166.7 PL=0
REFP 3 C00062 BC00062
CALL JOB:SEARCH-R1
IMOV P0056 V=23.0 PL=0
SET P0310 P0006
SFTON P0310
REFP 3 C00063 BC00063
CALL JOB:SEARCH-R1
SET P0310 P0006
SFTON P0310
MOVL C00064 BC00064 V=250.0 PL=0
SFTOF
MOVL C00065 BC00065 V=500.0
MOVL C00066 BC00066 V=166.7 PL=0
REFP 3 C00067 BC00067
CALL JOB:SEARCH-R1
IMOV P0056 V=23.0 PL=0
SET P0311 P0006
SFTON P0311
REFP 3 C00068 BC00068
CALL JOB:SEARCH-R1
SET P0311 P0006
SFTON P0311
MOVL C00069 BC00069 V=250.0 PL=0
SFTOF
MOVL C00070 BC00070 V=500.0
MOVL C00071 BC00071 V=500.0
MOVL C00072 BC00072 V=333.3
'------------------------
'W29.29
'------------------------
MOVL C00073 BC00073 V=166.7 PL=0
REFP 3 C00074 BC00074
CALL JOB:SEARCH-R1
IMOV P0056 V=23.0 PL=0
SET P0312 P0006
SFTON P0312
REFP 3 C00075 BC00075
CALL JOB:SEARCH-R1
SET P0312 P0006
SFTON P0312
MOVL C00076 BC00076 V=250.0 PL=0
SFTOF
'PRZEJAZD
MOVL C00077 BC00077 V=333.3
'PRZEJAZD
MOVL C00078 BC00078 V=500.0
MOVL C00079 BC00079 V=500.0
MOVL C00080 BC00080 V=333.3
MOVL C00081 BC00081 V=333.3
MOVL C00082 BC00082 V=166.7 PL=0
REFP 3 C00083 BC00083
CALL JOB:SEARCH-R1
IMOV P0056 V=23.0 PL=0
SET P0313 P0006
SFTON P0313
REFP 3 C00084 BC00084
CALL JOB:SEARCH-R1
SET P0313 P0006
SFTON P0313
MOVL C00085 BC00085 V=250.0 PL=0
SFTOF
MOVL C00086 BC00086 V=333.3
MOVL C00087 BC00087 V=166.7 PL=0
REFP 3 C00088 BC00088
CALL JOB:SEARCH-R1
IMOV P0056 V=23.0 PL=0
SET P0314 P0006
SFTON P0314
REFP 3 C00089 BC00089
CALL JOB:SEARCH-R1
SET P0314 P0006
SFTON P0314
MOVL C00090 BC00090 V=250.0 PL=0
SFTOF
MOVJ C00091 BC00091 VJ=10.00
MOVJ C00092 BC00092 VJ=10.00
MOVJ C00093 BC00093 VJ=30.00
MOVJ C00094 BC00094 VJ=20.00
MOVJ C00095 BC00095 VJ=50.00
MOVJ C00096 BC00096 VJ=20.00
MOVJ C00097 BC00097 VJ=10.00
MOVJ C00098 BC00098 VJ=20.00
MOVJ C00099 BC00099 VJ=20.00
'------------------------
'W28.2
'------------------------
MOVJ C00100 BC00100 VJ=10.00
MOVJ C00101 BC00101 VJ=10.00
MOVL C00102 BC00102 V=500.0
MOVL C00103 BC00103 V=500.0
'------------------------
'W62.5
'------------------------
MOVL C00104 BC00104 V=166.7 PL=0
REFP 3 C00105 BC00105
CALL JOB:SEARCH-R1
IMOV P0056 V=23.0 PL=0
SET P0351 P0006
SFTON P0351
REFP 3 C00106 BC00106
CALL JOB:SEARCH-R1
SET P0351 P0006
SFTON P0351
MOVL C00107 BC00107 V=250.0 PL=0
SFTOF
'PRZEJAZD
MOVL C00108 BC00108 V=500.0
MOVL C00109 BC00109 V=500.0
MOVL C00110 BC00110 V=500.0
MOVL C00111 BC00111 V=166.7 PL=0
REFP 3 C00112 BC00112
CALL JOB:SEARCH-R1
IMOV P0056 V=23.0 PL=0
SET P0352 P0006
SFTON P0352
REFP 3 C00113 BC00113
CALL JOB:SEARCH-R1
SET P0352 P0006
SFTON P0352
MOVL C00114 BC00114 V=250.0 PL=0
SFTOF
MOVL C00115 BC00115 V=500.0
'------------------------
'W29.8
'------------------------
MOVL C00116 BC00116 V=166.7 PL=0
REFP 3 C00117 BC00117
CALL JOB:SEARCH-R1
IMOV P0056 V=23.0 PL=0
SET P0353 P0006
SFTON P0353
REFP 3 C00118 BC00118
CALL JOB:SEARCH-R1
SET P0353 P0006
SFTON P0353
MOVL C00119 BC00119 V=250.0 PL=0
SFTOF
MOVL C00120 BC00120 V=500.0
'PRZEJAZD
MOVL C00121 BC00121 V=500.0
MOVJ C00122 BC00122 VJ=20.00
MOVL C00123 BC00123 V=500.0
MOVL C00124 BC00124 V=500.0
MOVL C00125 BC00125 V=500.0
'------------------------
'W29.11
'------------------------
MOVL C00126 BC00126 V=166.7 PL=0
REFP 3 C00127 BC00127
CALL JOB:SEARCH-R1
IMOV P0056 V=23.0 PL=0
SET P0354 P0006
SFTON P0354
REFP 3 C00128 BC00128
CALL JOB:SEARCH-R1
SET P0354 P0006
SFTON P0354
MOVL C00129 BC00129 V=250.0 PL=0
SFTOF
'PRZEJAZD
MOVL C00130 BC00130 V=500.0
'------------------------
'W29.14
'------------------------
MOVL C00131 BC00131 V=166.7 PL=0
REFP 3 C00132 BC00132
CALL JOB:SEARCH-R1
IMOV P0056 V=23.0 PL=0
SET P0355 P0006
SFTON P0355
REFP 3 C00133 BC00133
CALL JOB:SEARCH-R1
SET P0355 P0006
SFTON P0355
MOVL C00134 BC00134 V=250.0 PL=0
SFTOF
'PRZEJAZD
MOVL C00135 BC00135 V=500.0
'------------------------
'W63.17
'------------------------
MOVL C00136 BC00136 V=166.7 PL=0
REFP 3 C00137 BC00137
CALL JOB:SEARCH-R1
IMOV P0056 V=23.0 PL=0
SET P0356 P0006
SFTON P0356
REFP 3 C00138 BC00138
CALL JOB:SEARCH-R1
SET P0356 P0006
SFTON P0356
MOVL C00139 BC00139 V=250.0 PL=0
SFTOF
MOVL C00140 BC00140 V=500.0
MOVL C00141 BC00141 V=166.7 PL=0
REFP 3 C00142 BC00142
CALL JOB:SEARCH-R1
IMOV P0056 V=23.0 PL=0
SET P0357 P0006
SFTON P0357
REFP 3 C00143 BC00143
CALL JOB:SEARCH-R1
SET P0357 P0006
SFTON P0357
MOVL C00144 BC00144 V=250.0 PL=0
SFTOF
'PRZEJAZD
MOVL C00145 BC00145 V=500.0
MOVJ C00146 BC00146 VJ=30.00
MOVJ C00147 BC00147 VJ=30.00
MOVJ C00148 BC00148 VJ=30.00
MOVL C00149 BC00149 V=500.0
MOVL C00150 BC00150 V=500.0
'------------------------
'W62.20
'------------------------
MOVL C00151 BC00151 V=166.7 PL=0
REFP 3 C00152 BC00152
CALL JOB:SEARCH-R1
IMOV P0056 V=23.0 PL=0
SET P0358 P0006
SFTON P0358
REFP 3 C00153 BC00153
CALL JOB:SEARCH-R1
SET P0358 P0006
SFTON P0358
MOVL C00154 BC00154 V=250.0 PL=0
SFTOF
'PRZEJAZD
MOVL C00155 BC00155 V=500.0
'------------------------
'W63.23
'------------------------
MOVL C00156 BC00156 V=166.7 PL=0
REFP 3 C00157 BC00157
CALL JOB:SEARCH-R1
IMOV P0056 V=23.0 PL=0
SET P0359 P0006
SFTON P0359
REFP 3 C00158 BC00158
CALL JOB:SEARCH-R1
SET P0359 P0006
SFTON P0359
MOVL C00159 BC00159 V=250.0 PL=0
MOVL C00160 BC00160 V=500.0
'------------------------
'W29.29
'------------------------
MOVL C00161 BC00161 V=166.7 PL=0
REFP 3 C00162 BC00162
CALL JOB:SEARCH-R1
IMOV P0056 V=23.0 PL=0
SET P0360 P0006
SFTON P0360
REFP 3 C00163 BC00163
CALL JOB:SEARCH-R1
SET P0360 P0006
SFTON P0360
MOVL C00164 BC00164 V=250.0 PL=0
SFTOF
'PRZEJAZD
MOVL C00165 BC00165 V=500.0
MOVL C00166 BC00166 V=166.7 PL=0
REFP 3 C00167 BC00167
CALL JOB:SEARCH-R1
IMOV P0056 V=23.0 PL=0
SET P0361 P0006
SFTON P0361
REFP 3 C00168 BC00168
CALL JOB:SEARCH-R1
SET P0361 P0006
SFTON P0361
MOVL C00169 BC00169 V=250.0 PL=0
SFTOF
'------------------------
'W29.32
'------------------------
'PRZEJAZD
MOVL C00170 BC00170 V=500.0
MOVJ C00171 BC00171 VJ=10.00
MOVL C00172 BC00172 V=416.7
MOVL C00173 BC00173 V=166.7 PL=0
REFP 3 C00174 BC00174
CALL JOB:SEARCH-R1
IMOV P0056 V=23.0 PL=0
SET P0362 P0006
SFTON P0362
REFP 3 C00175 BC00175
CALL JOB:SEARCH-R1
SET P0362 P0006
SFTON P0362
MOVL C00176 BC00176 V=250.0 PL=0
SFTOF
MOVJ C00177 BC00177 VJ=20.00
MOVJ C00178 BC00178 VJ=30.00
MOVJ C00179 BC00179 VJ=15.00
MOVJ C00180 BC00180 VJ=15.00
MOVL C00181 BC00181 V=166.7
MOVL C00182 BC00182 V=166.7 PL=0
REFP 3 C00183 BC00183
CALL JOB:SEARCH-R1
IMOV P0056 V=23.0 PL=0
SET P0363 P0006
SFTON P0363
REFP 3 C00184 BC00184
CALL JOB:SEARCH-R1
SET P0363 P0006
SFTON P0363
MOVL C00185 BC00185 V=250.0 PL=0
SFTOF
MOVL C00186 BC00186 V=166.7 PL=0
REFP 3 C00187 BC00187
CALL JOB:SEARCH-R1
IMOV P0056 V=23.0 PL=0
SET P0364 P0006
SFTON P0364
REFP 3 C00188 BC00188
CALL JOB:SEARCH-R1
SET P0364 P0006
SFTON P0364
MOVL C00189 BC00189 V=250.0 PL=0
SFTOF
MOVJ C00190 BC00190 VJ=20.00
MOVJ C00191 BC00191 VJ=30.00
MOVJ C00192 BC00192 VJ=30.00
'KONIEC SEARCH WEW STRONA
MOVJ C00193 BC00193 VJ=30.00
MOVJ C00194 BC00194 VJ=20.00
MOVJ C00195 BC00195 VJ=10.00
MOVJ C00196 BC00196 VJ=20.00
MOVJ C00197 BC00197 VJ=20.00
'------------------------
'W29.2
'------------------------
MOVL C00198 BC00198 V=500.0
'------------------------
'W63.5
MACRO1 MJ#(0) ARGF9
'------------------------
SFTOF
SFTON P0301
MOVL C00199 BC00199 V=166.7 PL=0
ARCON
MOVL C00200 BC00200 V=10.0
ARCOF
SFTOF
MOVL C00201 BC00201 V=500.0
SFTON P0302
MOVL C00202 BC00202 V=166.7 PL=0
ARCON
MOVL C00203 BC00203 V=10.0
ARCOF
MOVL C00204 BC00204 V=166.7 PL=0
SFTOF
MOVL C00205 BC00205 V=500.0
SFTON P0303
MOVL C00206 BC00206 V=166.7 PL=0
ARCON
MOVL C00207 BC00207 V=10.0
ARCOF
SFTOF
MOVL C00208 BC00208 V=166.7 PL=0
MOVL C00209 BC00209 V=500.0
MOVJ C00210 BC00210 VJ=30.00
MOVJ C00211 BC00211 VJ=30.00
MOVJ C00212 BC00212 VJ=30.00
MOVL C00213 BC00213 V=500.0
'------------------------
'W29.14
'------------------------
SFTON P0304
MOVL C00214 BC00214 V=166.7 PL=0
ARCON
MOVL C00215 BC00215 V=10.0
ARCOF
MOVL C00216 BC00216 V=166.7 PL=0
SFTOF
'PRZEJAZD
MOVL C00217 BC00217 V=500.0
MOVL C00218 BC00218 V=500.0
'------------------------
'W63.17
'------------------------
SFTON P0305
MOVL C00219 BC00219 V=166.7 PL=0
ARCON
MOVL C00220 BC00220 V=10.0
ARCOF
MOVL C00221 BC00221 V=166.7 PL=0
SFTOF
MOVL C00222 BC00222 V=500.0
SFTON P0306
MOVL C00223 BC00223 V=166.7
ARCON
MOVL C00224 BC00224 V=10.0
ARCOF
MOVL C00225 BC00225 V=166.7 PL=0
SFTOF
'PRZEJAZD
MOVL C00226 BC00226 V=500.0
SFTON P0307
MOVL C00227 BC00227 V=166.7
ARCON
MOVL C00228 BC00228 V=10.0
ARCOF
MOVL C00229 BC00229 V=166.7 PL=0
SFTOF
MOVJ C00230 BC00230 VJ=20.00
MOVJ C00231 BC00231 VJ=20.00
MOVJ C00232 BC00232 VJ=30.00
MOVJ C00233 BC00233 VJ=30.00
MOVJ C00234 BC00234 VJ=30.00
MOVL C00235 BC00235 V=500.0
'------------------------
'W63.20
'------------------------
SFTON P0308
MOVL C00236 BC00236 V=166.7 PL=0
ARCON
MOVL C00237 BC00237 V=10.0
ARCOF
MOVL C00238 BC00238 V=166.7 PL=0
SFTOF
'PRZEJAZD
MOVL C00239 BC00239 V=500.0
'------------------------
'W63.23
'------------------------
SFTON P0309
MOVL C00240 BC00240 V=166.7 PL=0
ARCON
MOVL C00241 BC00241 V=10.0
ARCOF
MOVL C00242 BC00242 V=250.0 PL=0
SFTOF
MOVL C00243 BC00243 V=500.0
SFTON P0310
MOVL C00244 BC00244 V=166.7 PL=0
ARCON
MOVL C00245 BC00245 V=10.0
ARCOF
MOVL C00246 BC00246 V=250.0 PL=0
SFTOF
MOVL C00247 BC00247 V=500.0
SFTON P0311
MOVL C00248 BC00248 V=166.7 PL=0
ARCON
MOVL C00249 BC00249 V=10.0
ARCOF
MOVL C00250 BC00250 V=250.0 PL=0
SFTOF
MOVL C00251 BC00251 V=500.0
MOVL C00252 BC00252 V=500.0
MOVL C00253 BC00253 V=333.3
'------------------------
'W29.29
'------------------------
SFTON P0312
MOVL C00254 BC00254 V=166.7 PL=0
ARCON
MOVL C00255 BC00255 V=10.0
ARCOF
MOVL C00256 BC00256 V=250.0 PL=0
SFTOF
'PRZEJAZD
MOVL C00257 BC00257 V=333.3
'PRZEJAZD
'KONIEC SPAWANIA CZESCI WSPOLNEJ
MOVL C00258 BC00258 V=500.0
MOVL C00259 BC00259 V=500.0
MOVL C00260 BC00260 V=333.3
MOVL C00261 BC00261 V=333.3
SFTON P0313
MOVL C00262 BC00262 V=166.7 PL=0
ARCON
MOVL C00263 BC00263 V=10.0
ARCOF
MOVL C00264 BC00264 V=250.0 PL=0
SFTOF
MOVL C00265 BC00265 V=333.3
SFTON P0314
MOVL C00266 BC00266 V=166.7 PL=0
ARCON
MOVL C00267 BC00267 V=10.0
ARCOF
MOVL C00268 BC00268 V=250.0 PL=0
SFTOF
MOVJ C00269 BC00269 VJ=10.00
MOVJ C00270 BC00270 VJ=10.00
MOVJ C00271 BC00271 VJ=30.00
MOVJ C00272 BC00272 VJ=20.00
MOVJ C00273 BC00273 VJ=50.00
MOVJ C00274 BC00274 VJ=20.00
MOVJ C00275 BC00275 VJ=10.00
MOVJ C00276 BC00276 VJ=20.00
MOVJ C00277 BC00277 VJ=20.00
'------------------------
'W28.2
'------------------------
MOVJ C00278 BC00278 VJ=10.00
MOVJ C00279 BC00279 VJ=10.00
MOVL C00280 BC00280 V=500.0
MOVL C00281 BC00281 V=500.0
'------------------------
'W62.5
'------------------------
SFTON P0351
MOVL C00282 BC00282 V=166.7 PL=0
ARCON
MOVL C00283 BC00283 V=10.0
ARCOF
MOVL C00284 BC00284 V=250.0 PL=0
SFTOF
'PRZEJAZD
MOVL C00285 BC00285 V=500.0
MOVL C00286 BC00286 V=500.0
MOVL C00287 BC00287 V=500.0
SFTON P0352
MOVL C00288 BC00288 V=166.7 PL=0
ARCON
MOVL C00289 BC00289 V=10.0
ARCOF
MOVL C00290 BC00290 V=250.0 PL=0
SFTOF
MOVL C00291 BC00291 V=500.0
'------------------------
'W29.8
'------------------------
SFTON P0353
MOVL C00292 BC00292 V=166.7 PL=0
ARCON
MOVL C00293 BC00293 V=10.0
ARCOF
MOVL C00294 BC00294 V=250.0 PL=0
SFTOF
MOVL C00295 BC00295 V=500.0
'PRZEJAZD
MOVL C00296 BC00296 V=500.0
MOVJ C00297 BC00297 VJ=20.00
MOVL C00298 BC00298 V=500.0
MOVL C00299 BC00299 V=500.0
MOVL C00300 BC00300 V=500.0
'------------------------
'W29.11
'------------------------
SFTON P0354
MOVL C00301 BC00301 V=166.7 PL=0
ARCON
MOVL C00302 BC00302 V=10.0
ARCOF
MOVL C00303 BC00303 V=250.0 PL=0
SFTOF
'PRZEJAZD
MOVL C00304 BC00304 V=500.0
'------------------------
'W29.14
'------------------------
SFTON P0355
MOVL C00305 BC00305 V=166.7 PL=0
ARCON
MOVL C00306 BC00306 V=10.0
ARCOF
MOVL C00307 BC00307 V=250.0 PL=0
SFTOF
'PRZEJAZD
MOVL C00308 BC00308 V=500.0
'------------------------
'W63.17
'------------------------
SFTON P0356
MOVL C00309 BC00309 V=166.7 PL=0
ARCON
MOVL C00310 BC00310 V=10.0
ARCOF
MOVL C00311 BC00311 V=250.0 PL=0
SFTOF
MOVL C00312 BC00312 V=500.0
SFTON P0357
MOVL C00313 BC00313 V=166.7 PL=0
ARCON
MOVL C00314 BC00314 V=10.0
ARCOF
MOVL C00315 BC00315 V=250.0 PL=0
SFTOF
'PRZEJAZD
MOVL C00316 BC00316 V=500.0
MOVJ C00317 BC00317 VJ=30.00
MOVJ C00318 BC00318 VJ=30.00
MOVJ C00319 BC00319 VJ=30.00
MOVL C00320 BC00320 V=500.0
MOVL C00321 BC00321 V=500.0
'------------------------
'W62.20
'------------------------
SFTON P0358
MOVL C00322 BC00322 V=166.7 PL=0
ARCON
MOVL C00323 BC00323 V=10.0
ARCOF
MOVL C00324 BC00324 V=250.0 PL=0
SFTOF
'PRZEJAZD
MOVL C00325 BC00325 V=500.0
'------------------------
'W63.23
'------------------------
SFTON P0359
MOVL C00326 BC00326 V=166.7 PL=0
ARCON
MOVL C00327 BC00327 V=10.0
ARCOF
MOVL C00328 BC00328 V=250.0 PL=0
MOVL C00329 BC00329 V=500.0
'------------------------
'W29.29
'------------------------
SFTON P0360
MOVL C00330 BC00330 V=166.7 PL=0
ARCON
MOVL C00331 BC00331 V=10.0
ARCOF
MOVL C00332 BC00332 V=250.0 PL=0
SFTOF
'PRZEJAZD
MOVL C00333 BC00333 V=500.0
SFTON P0361
MOVL C00334 BC00334 V=166.7 PL=0
ARCON
MOVL C00335 BC00335 V=10.0
ARCOF
MOVL C00336 BC00336 V=250.0 PL=0
SFTOF
'------------------------
'W29.32
'------------------------
'PRZEJAZD
MOVL C00337 BC00337 V=500.0
MOVJ C00338 BC00338 VJ=10.00
MOVL C00339 BC00339 V=416.7
SFTON P0362
MOVL C00340 BC00340 V=166.7 PL=0
ARCON
MOVL C00341 BC00341 V=10.0
ARCOF
MOVL C00342 BC00342 V=250.0 PL=0
SFTOF
MOVJ C00343 BC00343 VJ=20.00
MOVJ C00344 BC00344 VJ=30.00
MOVJ C00345 BC00345 VJ=15.00
MOVJ C00346 BC00346 VJ=15.00
MOVL C00347 BC00347 V=166.7
SFTON P0363
MOVL C00348 BC00348 V=166.7 PL=0
ARCON
MOVL C00349 BC00349 V=10.0
ARCOF
MOVL C00350 BC00350 V=250.0 PL=0
SFTOF
SFTON P0364
MOVL C00351 BC00351 V=166.7 PL=0
ARCON
MOVL C00352 BC00352 V=10.0
ARCOF
MOVL C00353 BC00353 V=250.0 PL=0
SFTOF
MOVJ C00354 BC00354 VJ=20.00
MOVJ C00355 BC00355 VJ=30.00
MOVJ C00356 BC00356 VJ=30.00
CALL JOB:MOVE_OUT_OF_TUNNEL
CALL JOB:CLEAN-R1
CALL JOB:MOVE_INTO_TUNNEL
'KONIEC SPAWANIA WEW STRONA
MOVJ C00357 BC00357 VJ=10.00
MOVJ C00358 BC00358 VJ=10.00
MOVJ C00359 BC00359 VJ=20.00
MOVJ C00360 BC00360 VJ=20.00
MOVJ C00361 BC00361 VJ=10.00
MOVJ C00362 BC00362 VJ=10.00
'------------------------
'W29.2
'------------------------
MOVL C00363 BC00363 V=500.0
'------------------------
'W63.5
'------------------------
SFTOF
MOVL C00364 BC00364 V=166.7 PL=0
REFP 3 C00365 BC00365
CALL JOB:SEARCH-R1
IMOV P0056 V=50.0 PL=0
SET P0301 P0006
SFTON P0301
REFP 3 C00366 BC00366
CALL JOB:SEARCH-R1
SET P0301 P0006
SFTON P0301
MOVL C00367 BC00367 V=166.7 PL=0
SFTOF
MOVL C00368 BC00368 V=500.0
MOVL C00369 BC00369 V=166.7 PL=0
REFP 3 C00370 BC00370
CALL JOB:SEARCH-R1
IMOV P0056 V=50.0 PL=0
SET P0302 P0006
SFTON P0302
REFP 3 C00371 BC00371
CALL JOB:SEARCH-R1
SET P0302 P0006
SFTON P0302
MOVL C00372 BC00372 V=166.7 PL=0
SFTOF
MOVL C00373 BC00373 V=500.0
MOVL C00374 BC00374 V=166.7 PL=0
REFP 3 C00375 BC00375
CALL JOB:SEARCH-R1
IMOV P0056 V=50.0 PL=0
SET P0303 P0006
SFTON P0303
REFP 3 C00376 BC00376
CALL JOB:SEARCH-R1
SET P0303 P0006
SFTON P0303
SFTOF
MOVL C00377 BC00377 V=166.7 PL=0
MOVL C00378 BC00378 V=500.0
MOVJ C00379 BC00379 VJ=30.00
MOVJ C00380 BC00380 VJ=30.00
MOVJ C00381 BC00381 VJ=20.00
MOVJ C00382 BC00382 VJ=30.00
MOVL C00383 BC00383 V=500.0
'------------------------
'W29.14
'------------------------
MOVL C00384 BC00384 V=166.7 PL=0
REFP 3 C00385 BC00385
CALL JOB:SEARCH-R1
IMOV P0056 V=23.0 PL=0
SET P0304 P0006
SFTON P0304
REFP 3 C00386 BC00386
CALL JOB:SEARCH-R1
SET P0304 P0006
SFTON P0304
MOVL C00387 BC00387 V=66.7 PL=0
SFTOF
'PRZEJAZD
MOVL C00388 BC00388 V=500.0
MOVL C00389 BC00389 V=500.0
'------------------------
'W63.17
'------------------------
MOVL C00390 BC00390 V=166.7 PL=0
REFP 3 C00391 BC00391
CALL JOB:SEARCH-R1
IMOV P0056 V=23.0 PL=0
SET P0305 P0006
SFTON P0305
REFP 3 C00392 BC00392
CALL JOB:SEARCH-R1
SET P0305 P0006
SFTON P0305
MOVL C00393 BC00393 V=166.7 PL=0
SFTOF
MOVL C00394 BC00394 V=500.0
MOVL C00395 BC00395 V=166.7
REFP 3 C00396 BC00396
CALL JOB:SEARCH-R1
IMOV P0056 V=23.0 PL=0
SET P0306 P0006
SFTON P0306
REFP 3 C00397 BC00397
CALL JOB:SEARCH-R1
SET P0306 P0006
SFTON P0306
MOVL C00398 BC00398 V=166.7 PL=0
'PRZEJAZD
MOVL C00399 BC00399 V=500.0
MOVL C00400 BC00400 V=166.7
REFP 3 C00401 BC00401
CALL JOB:SEARCH-R1
IMOV P0056 V=23.0 PL=0
SET P0307 P0006
SFTON P0307
REFP 3 C00402 BC00402
CALL JOB:SEARCH-R1
SET P0307 P0006
SFTON P0307
MOVL C00403 BC00403 V=166.7 PL=0
SFTOF
MOVJ C00404 BC00404 VJ=20.00
MOVJ C00405 BC00405 VJ=20.00
MOVJ C00406 BC00406 VJ=30.00
MOVJ C00407 BC00407 VJ=30.00
MOVL C00408 BC00408 V=500.0
'------------------------
'W63.20
'------------------------
MOVL C00409 BC00409 V=166.7 PL=0
REFP 3 C00410 BC00410
CALL JOB:SEARCH-R1
IMOV P0056 V=23.0 PL=0
SET P0308 P0006
SFTON P0308
REFP 3 C00411 BC00411
CALL JOB:SEARCH-R1
SET P0308 P0006
SFTON P0308
MOVL C00412 BC00412 V=166.7 PL=0
SFTOF
'PRZEJAZD
MOVL C00413 BC00413 V=500.0
'------------------------
'W63.23
'------------------------
MOVL C00414 BC00414 V=166.7 PL=0
REFP 3 C00415 BC00415
CALL JOB:SEARCH-R1
IMOV P0056 V=23.0 PL=0
SET P0309 P0006
SFTON P0309
REFP 3 C00416 BC00416
CALL JOB:SEARCH-R1
SET P0309 P0006
SFTON P0309
MOVL C00417 BC00417 V=250.0 PL=0
SFTOF
MOVL C00418 BC00418 V=500.0
MOVL C00419 BC00419 V=166.7 PL=0
REFP 3 C00420 BC00420
CALL JOB:SEARCH-R1
IMOV P0056 V=23.0 PL=0
SET P0310 P0006
SFTON P0310
REFP 3 C00421 BC00421
CALL JOB:SEARCH-R1
SET P0310 P0006
SFTON P0310
MOVL C00422 BC00422 V=250.0 PL=0
SFTOF
MOVL C00423 BC00423 V=500.0
MOVL C00424 BC00424 V=166.7 PL=0
REFP 3 C00425 BC00425
CALL JOB:SEARCH-R1
IMOV P0056 V=23.0 PL=0
SET P0311 P0006
SFTON P0311
REFP 3 C00426 BC00426
CALL JOB:SEARCH-R1
SET P0311 P0006
SFTON P0311
MOVL C00427 BC00427 V=250.0 PL=0
SFTOF
MOVL C00428 BC00428 V=500.0
MOVL C00429 BC00429 V=500.0
MOVL C00430 BC00430 V=500.0
MOVL C00431 BC00431 V=333.3
'------------------------
'W29.29
'------------------------
MOVL C00432 BC00432 V=166.7 PL=0
REFP 3 C00433 BC00433
CALL JOB:SEARCH-R1
IMOV P0056 V=23.0 PL=0
SET P0312 P0006
SFTON P0312
REFP 3 C00434 BC00434
CALL JOB:SEARCH-R1
SET P0312 P0006
SFTON P0312
MOVL C00435 BC00435 V=250.0 PL=0
SFTOF
'PRZEJAZD
MOVL C00436 BC00436 V=333.3
'PRZEJAZD
MOVL C00437 BC00437 V=500.0
MOVL C00438 BC00438 V=500.0
MOVL C00439 BC00439 V=333.3
MOVL C00440 BC00440 V=333.3
MOVL C00441 BC00441 V=166.7 PL=0
REFP 3 C00442 BC00442
CALL JOB:SEARCH-R1
IMOV P0056 V=23.0 PL=0
SET P0313 P0006
SFTON P0313
REFP 3 C00443 BC00443
CALL JOB:SEARCH-R1
SET P0313 P0006
SFTON P0313
MOVL C00444 BC00444 V=250.0 PL=0
SFTOF
MOVL C00445 BC00445 V=333.3
MOVL C00446 BC00446 V=166.7 PL=0
REFP 3 C00447 BC00447
CALL JOB:SEARCH-R1
IMOV P0056 V=23.0 PL=0
SET P0314 P0006
SFTON P0314
REFP 3 C00448 BC00448
CALL JOB:SEARCH-R1
SET P0314 P0006
SFTON P0314
MOVL C00449 BC00449 V=250.0 PL=0
SFTOF
MOVJ C00450 BC00450 VJ=10.00
MOVJ C00451 BC00451 VJ=10.00
MOVJ C00452 BC00452 VJ=20.00
MOVJ C00453 BC00453 VJ=50.00
MOVJ C00454 BC00454 VJ=20.00
MOVJ C00455 BC00455 VJ=10.00
'------------------------
'W28.2
'------------------------
MOVJ C00456 BC00456 VJ=10.00
MOVJ C00457 BC00457 VJ=10.00
MOVL C00458 BC00458 V=500.0
MOVL C00459 BC00459 V=500.0
'------------------------
'W62.5
'------------------------
MOVL C00460 BC00460 V=166.7 PL=0
REFP 3 C00461 BC00461
CALL JOB:SEARCH-R1
IMOV P0056 V=23.0 PL=0
SET P0351 P0006
SFTON P0351
REFP 3 C00462 BC00462
CALL JOB:SEARCH-R1
SET P0351 P0006
SFTON P0351
MOVL C00463 BC00463 V=250.0 PL=0
SFTOF
'PRZEJAZD
MOVL C00464 BC00464 V=500.0
MOVL C00465 BC00465 V=500.0
MOVL C00466 BC00466 V=500.0
MOVL C00467 BC00467 V=166.7 PL=0
REFP 3 C00468 BC00468
CALL JOB:SEARCH-R1
IMOV P0056 V=23.0 PL=0
SET P0352 P0006
SFTON P0352
REFP 3 C00469 BC00469
CALL JOB:SEARCH-R1
SET P0352 P0006
SFTON P0352
MOVL C00470 BC00470 V=250.0 PL=0
SFTOF
MOVL C00471 BC00471 V=500.0
'------------------------
'W29.8
'------------------------
MOVL C00472 BC00472 V=166.7 PL=0
REFP 3 C00473 BC00473
CALL JOB:SEARCH-R1
IMOV P0056 V=23.0 PL=0
SET P0353 P0006
SFTON P0353
REFP 3 C00474 BC00474
CALL JOB:SEARCH-R1
SET P0353 P0006
SFTON P0353
MOVL C00475 BC00475 V=250.0 PL=0
SFTOF
MOVL C00476 BC00476 V=500.0
'PRZEJAZD
MOVL C00477 BC00477 V=500.0
MOVJ C00478 BC00478 VJ=20.00
MOVJ C00479 BC00479 VJ=20.00
MOVL C00480 BC00480 V=500.0
MOVL C00481 BC00481 V=500.0
MOVL C00482 BC00482 V=500.0
'------------------------
'W29.11
'------------------------
MOVL C00483 BC00483 V=166.7 PL=0
REFP 3 C00484 BC00484
CALL JOB:SEARCH-R1
IMOV P0056 V=23.0 PL=0
SET P0354 P0006
SFTON P0354
REFP 3 C00485 BC00485
CALL JOB:SEARCH-R1
SET P0354 P0006
SFTON P0354
MOVL C00486 BC00486 V=250.0 PL=0
SFTOF
'PRZEJAZD
MOVL C00487 BC00487 V=500.0
'------------------------
'W29.14
'------------------------
MOVL C00488 BC00488 V=166.7 PL=0
REFP 3 C00489 BC00489
CALL JOB:SEARCH-R1
IMOV P0056 V=23.0 PL=0
SET P0355 P0006
SFTON P0355
REFP 3 C00490 BC00490
CALL JOB:SEARCH-R1
SET P0355 P0006
SFTON P0355
MOVL C00491 BC00491 V=250.0 PL=0
SFTOF
'PRZEJAZD
MOVL C00492 BC00492 V=500.0
'------------------------
'W63.17
'------------------------
MOVL C00493 BC00493 V=166.7 PL=0
REFP 3 C00494 BC00494
CALL JOB:SEARCH-R1
IMOV P0056 V=23.0 PL=0
SET P0356 P0006
SFTON P0356
REFP 3 C00495 BC00495
CALL JOB:SEARCH-R1
SET P0356 P0006
SFTON P0356
MOVL C00496 BC00496 V=250.0 PL=0
SFTOF
MOVL C00497 BC00497 V=500.0
MOVL C00498 BC00498 V=166.7 PL=0
REFP 3 C00499 BC00499
CALL JOB:SEARCH-R1
IMOV P0056 V=23.0 PL=0
SET P0357 P0006
SFTON P0357
REFP 3 C00500 BC00500
CALL JOB:SEARCH-R1
SET P0357 P0006
SFTON P0357
MOVL C00501 BC00501 V=250.0 PL=0
SFTOF
'PRZEJAZD
MOVL C00502 BC00502 V=500.0
MOVJ C00503 BC00503 VJ=30.00
MOVJ C00504 BC00504 VJ=30.00
MOVL C00505 BC00505 V=500.0
MOVL C00506 BC00506 V=500.0
'------------------------
'W62.20
'------------------------
MOVL C00507 BC00507 V=166.7 PL=0
REFP 3 C00508 BC00508
CALL JOB:SEARCH-R1
IMOV P0056 V=23.0 PL=0
SET P0358 P0006
SFTON P0358
REFP 3 C00509 BC00509
CALL JOB:SEARCH-R1
SET P0358 P0006
SFTON P0358
MOVL C00510 BC00510 V=250.0 PL=0
SFTOF
'PRZEJAZD
MOVL C00511 BC00511 V=500.0
'------------------------
'W63.23
'------------------------
MOVL C00512 BC00512 V=166.7 PL=0
REFP 3 C00513 BC00513
CALL JOB:SEARCH-R1
IMOV P0056 V=23.0 PL=0
SET P0359 P0006
SFTON P0359
REFP 3 C00514 BC00514
CALL JOB:SEARCH-R1
SET P0359 P0006
SFTON P0359
MOVL C00515 BC00515 V=250.0 PL=0
MOVL C00516 BC00516 V=500.0
'------------------------
'W29.29
'------------------------
MOVL C00517 BC00517 V=166.7 PL=0
REFP 3 C00518 BC00518
CALL JOB:SEARCH-R1
IMOV P0056 V=23.0 PL=0
SET P0360 P0006
SFTON P0360
REFP 3 C00519 BC00519
CALL JOB:SEARCH-R1
SET P0360 P0006
SFTON P0360
MOVL C00520 BC00520 V=250.0 PL=0
SFTOF
'PRZEJAZD
MOVL C00521 BC00521 V=500.0
MOVL C00522 BC00522 V=166.7 PL=0
REFP 3 C00523 BC00523
CALL JOB:SEARCH-R1
IMOV P0056 V=23.0 PL=0
SET P0361 P0006
SFTON P0361
REFP 3 C00524 BC00524
CALL JOB:SEARCH-R1
SET P0361 P0006
SFTON P0361
MOVL C00525 BC00525 V=250.0 PL=0
SFTOF
'------------------------
'W29.32
'------------------------
'PRZEJAZD
MOVL C00526 BC00526 V=500.0
MOVJ C00527 BC00527 VJ=10.00
MOVL C00528 BC00528 V=416.7
MOVL C00529 BC00529 V=166.7 PL=0
REFP 3 C00530 BC00530
CALL JOB:SEARCH-R1
IMOV P0056 V=23.0 PL=0
SET P0362 P0006
SFTON P0362
REFP 3 C00531 BC00531
CALL JOB:SEARCH-R1
SET P0362 P0006
SFTON P0362
MOVL C00532 BC00532 V=250.0 PL=0
SFTOF
MOVJ C00533 BC00533 VJ=20.00
MOVJ C00534 BC00534 VJ=30.00
MOVJ C00535 BC00535 VJ=15.00
MOVJ C00536 BC00536 VJ=15.00
MOVL C00537 BC00537 V=166.7
MOVL C00538 BC00538 V=166.7 PL=0
REFP 3 C00539 BC00539
CALL JOB:SEARCH-R1
IMOV P0056 V=23.0 PL=0
SET P0363 P0006
SFTON P0363
REFP 3 C00540 BC00540
CALL JOB:SEARCH-R1
SET P0363 P0006
SFTON P0363
MOVL C00541 BC00541 V=250.0 PL=0
SFTOF
MOVL C00542 BC00542 V=166.7 PL=0
REFP 3 C00543 BC00543
CALL JOB:SEARCH-R1
IMOV P0056 V=23.0 PL=0
SET P0364 P0006
SFTON P0364
REFP 3 C00544 BC00544
CALL JOB:SEARCH-R1
SET P0364 P0006
SFTON P0364
MOVL C00545 BC00545 V=250.0 PL=0
SFTOF
MOVJ C00546 BC00546 VJ=20.00
MOVJ C00547 BC00547 VJ=30.00
MOVJ C00548 BC00548 VJ=30.00
'KONIEC SEARCH WEW STRONA
MOVJ C00549 BC00549 VJ=30.00
MOVJ C00550 BC00550 VJ=20.00
MOVJ C00551 BC00551 VJ=10.00
MOVJ C00552 BC00552 VJ=20.00
MOVJ C00553 BC00553 VJ=20.00
'------------------------
'W29.2
'------------------------
MOVL C00554 BC00554 V=500.0
'------------------------
'W63.5
MACRO1 MJ#(0) ARGF9
'------------------------
SFTOF
SFTON P0301
MOVL C00555 BC00555 V=166.7 PL=0
ARCON
MOVL C00556 BC00556 V=8.3
ARCOF
SFTOF
MOVL C00557 BC00557 V=500.0
MACRO1 MJ#(0) ARGF24
SFTON P0302
MOVL C00558 BC00558 V=166.7 PL=0
ARCON
MOVL C00559 BC00559 V=8.3
ARCOF
MOVL C00560 BC00560 V=166.7 PL=0
SFTOF
MOVL C00561 BC00561 V=500.0
SFTON P0303
MOVL C00562 BC00562 V=166.7 PL=0
ARCON
MOVL C00563 BC00563 V=8.3
ARCOF
SFTOF
MOVL C00564 BC00564 V=166.7 PL=0
MOVL C00565 BC00565 V=500.0
MOVJ C00566 BC00566 VJ=30.00
MOVJ C00567 BC00567 VJ=20.00
MOVJ C00568 BC00568 VJ=30.00
MOVJ C00569 BC00569 VJ=30.00
MOVL C00570 BC00570 V=500.0
'------------------------
'W29.14
'------------------------
SFTON P0304
MOVL C00571 BC00571 V=166.7 PL=0
ARCON
MOVL C00572 BC00572 V=8.3
ARCOF
MOVL C00573 BC00573 V=166.7 PL=0
SFTOF
'PRZEJAZD
MOVL C00574 BC00574 V=500.0
MOVL C00575 BC00575 V=500.0
'------------------------
'W63.17
'------------------------
SFTON P0305
MOVL C00576 BC00576 V=166.7 PL=0
ARCON
MOVL C00577 BC00577 V=8.3
ARCOF
MOVL C00578 BC00578 V=166.7 PL=0
SFTOF
MOVL C00579 BC00579 V=500.0
SFTON P0306
MOVL C00580 BC00580 V=166.7
ARCON
MOVL C00581 BC00581 V=8.3
ARCOF
MOVL C00582 BC00582 V=166.7 PL=0
SFTOF
'PRZEJAZD
MOVL C00583 BC00583 V=500.0
SFTON P0307
MOVL C00584 BC00584 V=166.7
ARCON
MOVL C00585 BC00585 V=8.3
ARCOF
MOVL C00586 BC00586 V=166.7 PL=0
SFTOF
MOVJ C00587 BC00587 VJ=20.00
MOVJ C00588 BC00588 VJ=20.00
MOVJ C00589 BC00589 VJ=30.00
MOVJ C00590 BC00590 VJ=30.00
MOVL C00591 BC00591 V=500.0
'------------------------
'W63.20
'------------------------
SFTON P0308
MOVL C00592 BC00592 V=166.7 PL=0
ARCON
MOVL C00593 BC00593 V=8.3
ARCOF
MOVL C00594 BC00594 V=166.7 PL=0
SFTOF
'PRZEJAZD
MOVL C00595 BC00595 V=500.0
'------------------------
'W63.23
'------------------------
SFTON P0309
MOVL C00596 BC00596 V=166.7 PL=0
ARCON
MOVL C00597 BC00597 V=8.3
ARCOF
MOVL C00598 BC00598 V=250.0 PL=0
SFTOF
MOVL C00599 BC00599 V=500.0
SFTON P0310
MOVL C00600 BC00600 V=166.7 PL=0
ARCON
MOVL C00601 BC00601 V=8.3
ARCOF
MOVL C00602 BC00602 V=250.0 PL=0
SFTOF
MOVL C00603 BC00603 V=500.0
SFTON P0311
MOVL C00604 BC00604 V=166.7 PL=0
ARCON
MOVL C00605 BC00605 V=8.3
ARCOF
MOVL C00606 BC00606 V=250.0 PL=0
SFTOF
MOVL C00607 BC00607 V=500.0
MOVL C00608 BC00608 V=500.0
MOVL C00609 BC00609 V=333.3
'------------------------
'W29.29
'------------------------
SFTON P0312
MOVL C00610 BC00610 V=166.7 PL=0
ARCON
MOVL C00611 BC00611 V=8.3
ARCOF
MOVL C00612 BC00612 V=250.0 PL=0
SFTOF
'PRZEJAZD
MOVL C00613 BC00613 V=333.3
'PRZEJAZD
'KONIEC SPAWANIA CZESCI WSPOLNEJ
MOVL C00614 BC00614 V=500.0
MOVL C00615 BC00615 V=500.0
MOVL C00616 BC00616 V=500.0
MOVL C00617 BC00617 V=333.3
MOVL C00618 BC00618 V=333.3
SFTON P0313
MOVL C00619 BC00619 V=166.7 PL=0
ARCON
MOVL C00620 BC00620 V=8.3
ARCOF
MOVL C00621 BC00621 V=250.0 PL=0
SFTOF
MOVL C00622 BC00622 V=333.3
SFTON P0314
MOVL C00623 BC00623 V=166.7 PL=0
ARCON
MOVL C00624 BC00624 V=8.3
ARCOF
MOVL C00625 BC00625 V=250.0 PL=0
SFTOF
MOVJ C00626 BC00626 VJ=10.00
MOVJ C00627 BC00627 VJ=10.00
MOVJ C00628 BC00628 VJ=30.00
MOVJ C00629 BC00629 VJ=20.00
MOVJ C00630 BC00630 VJ=50.00
MOVJ C00631 BC00631 VJ=20.00
MOVJ C00632 BC00632 VJ=10.00
MOVJ C00633 BC00633 VJ=20.00
MOVJ C00634 BC00634 VJ=20.00
'------------------------
'W28.2
'------------------------
MOVJ C00635 BC00635 VJ=10.00
MOVJ C00636 BC00636 VJ=10.00
MOVL C00637 BC00637 V=500.0
MOVL C00638 BC00638 V=500.0
'------------------------
'W62.5
'------------------------
SFTON P0351
MOVL C00639 BC00639 V=166.7 PL=0
ARCON
MOVL C00640 BC00640 V=8.3
ARCOF
MOVL C00641 BC00641 V=250.0 PL=0
SFTOF
'PRZEJAZD
MOVL C00642 BC00642 V=500.0
MOVL C00643 BC00643 V=500.0
MOVL C00644 BC00644 V=500.0
SFTON P0352
MOVL C00645 BC00645 V=166.7 PL=0
ARCON
MOVL C00646 BC00646 V=8.3
ARCOF
MOVL C00647 BC00647 V=250.0 PL=0
SFTOF
MOVL C00648 BC00648 V=500.0
'------------------------
'W29.8
'------------------------
SFTON P0353
MOVL C00649 BC00649 V=166.7 PL=0
ARCON
MOVL C00650 BC00650 V=8.3
ARCOF
MOVL C00651 BC00651 V=250.0 PL=0
SFTOF
MOVL C00652 BC00652 V=500.0
'PRZEJAZD
MOVL C00653 BC00653 V=500.0
MOVJ C00654 BC00654 VJ=20.00
MOVL C00655 BC00655 V=500.0
MOVL C00656 BC00656 V=500.0
MOVL C00657 BC00657 V=500.0
'------------------------
'W29.11
'------------------------
SFTON P0354
MOVL C00658 BC00658 V=166.7 PL=0
ARCON
MOVL C00659 BC00659 V=8.3
ARCOF
MOVL C00660 BC00660 V=250.0 PL=0
SFTOF
'PRZEJAZD
MOVL C00661 BC00661 V=500.0
'------------------------
'W29.14
'------------------------
SFTON P0355
MOVL C00662 BC00662 V=166.7 PL=0
ARCON
MOVL C00663 BC00663 V=8.3
ARCOF
MOVL C00664 BC00664 V=250.0 PL=0
SFTOF
'PRZEJAZD
MOVL C00665 BC00665 V=500.0
'------------------------
'W63.17
'------------------------
SFTON P0356
MOVL C00666 BC00666 V=166.7 PL=0
ARCON
MOVL C00667 BC00667 V=8.3
ARCOF
MOVL C00668 BC00668 V=250.0 PL=0
SFTOF
MOVL C00669 BC00669 V=500.0
SFTON P0357
MOVL C00670 BC00670 V=166.7 PL=0
ARCON
MOVL C00671 BC00671 V=8.3
ARCOF
MOVL C00672 BC00672 V=250.0 PL=0
SFTOF
'PRZEJAZD
MOVL C00673 BC00673 V=500.0
MOVJ C00674 BC00674 VJ=30.00
MOVJ C00675 BC00675 VJ=30.00
MOVJ C00676 BC00676 VJ=30.00
MOVL C00677 BC00677 V=500.0
MOVL C00678 BC00678 V=500.0
'------------------------
'W62.20
'------------------------
SFTON P0358
MOVL C00679 BC00679 V=166.7 PL=0
ARCON
MOVL C00680 BC00680 V=8.3
ARCOF
MOVL C00681 BC00681 V=250.0 PL=0
SFTOF
'PRZEJAZD
MOVL C00682 BC00682 V=500.0
'------------------------
'W63.23
'------------------------
SFTON P0359
MOVL C00683 BC00683 V=166.7 PL=0
ARCON
MOVL C00684 BC00684 V=8.3
ARCOF
MOVL C00685 BC00685 V=250.0 PL=0
MOVL C00686 BC00686 V=500.0
'------------------------
'W29.29
'------------------------
SFTON P0360
MOVL C00687 BC00687 V=166.7 PL=0
ARCON
MOVL C00688 BC00688 V=8.3
ARCOF
MOVL C00689 BC00689 V=250.0 PL=0
SFTOF
'PRZEJAZD
MOVL C00690 BC00690 V=500.0
SFTON P0361
MOVL C00691 BC00691 V=166.7 PL=0
ARCON
MOVL C00692 BC00692 V=8.3
ARCOF
MOVL C00693 BC00693 V=250.0 PL=0
SFTOF
'------------------------
'W29.32
'------------------------
'PRZEJAZD
MOVL C00694 BC00694 V=500.0
MOVJ C00695 BC00695 VJ=10.00
MOVL C00696 BC00696 V=416.7
SFTON P0362
MOVL C00697 BC00697 V=166.7 PL=0
ARCON
MOVL C00698 BC00698 V=8.3
ARCOF
MOVL C00699 BC00699 V=250.0 PL=0
SFTOF
MOVJ C00700 BC00700 VJ=20.00
MOVJ C00701 BC00701 VJ=30.00
MOVJ C00702 BC00702 VJ=15.00
MOVJ C00703 BC00703 VJ=15.00
MOVL C00704 BC00704 V=166.7
SFTON P0363
MOVL C00705 BC00705 V=166.7 PL=0
ARCON
MOVL C00706 BC00706 V=8.3
ARCOF
MOVL C00707 BC00707 V=250.0 PL=0
SFTOF
SFTON P0364
MOVL C00708 BC00708 V=166.7 PL=0
ARCON
MOVL C00709 BC00709 V=8.3
ARCOF
MOVL C00710 BC00710 V=250.0 PL=0
SFTOF
MOVJ C00711 BC00711 VJ=20.00
MOVJ C00712 BC00712 VJ=30.00
MOVJ C00713 BC00713 VJ=30.00
CALL JOB:MOVE_OUT_OF_TUNNEL
END
